(* POU Stations/ST_03_Ruestsaetze/ST_03_PRGs/ST03_Init_AbholPos, ST *)
PROGRAM ST03_Init_AbholPos
VAR
	RoboPos31		:BOOL;
	RoboPos35		:BOOL;
	RoboPosErr		:BOOL;
	CamDone			:BOOL;
	fb_Ton_PosErr	:TON;

	MsgOK			: BOOL;
END_VAR
(* Hier werden alle Abholpositionen am Rüstsatz bestimmt.
Ausnahmen:
	alte Rüstsätze:
		P360 74pol 
		P379 91pol 
		P489 168pol
		P4992 35pol
	Tampondrucker:
		P312 93pol
		P4991 102pol			*)

RoboPos31:=FALSE;
RoboPos35:=FALSE;
RoboPosErr:=FALSE;
CASE  gTypeCode OF

360,489:	(*74polig, 91polig, 168polig*)

	RoboPos31:=TRUE;

379: (*91 pol*)
RoboPos31:=
		ST08_412_B59_0.BitInToCheck;
	ST03_Main.Result:=RESULT_OK;		(* immer OK, wenn es keine Prüfung gibt*)

4992: (*35polig*)
	RoboPos31:=
		NOT ST08_412_B58_5_35pol.BitInToCheck AND	(*links*)
		ST08_412_B58_6_35pol.BitInToCheck;			(*rechts*)
	RoboPos35:=
		ST08_412_B58_5_35pol.BitInToCheck AND		(*links*)
		NOT ST08_412_B58_6_35pol.BitInToCheck;		(*rechts*)
	RoboPosErr:=
		ST08_412_B58_5_35pol.BitInToCheck AND		(*links*)
		ST08_412_B58_6_35pol.BitInToCheck;			(*rechts*)
	ST03_Main.Result:=RESULT_OK;		(* immer OK, wenn es keine Prüfung gibt*)

4871:(*154polig*)
	RoboPos31:=
		ST03_426_B68_4.BitInToCheck; 		(* Zuführung ISK auf Übergabeposition Robo Palettierer*)
	ST03_Main.Result:=RESULT_OK;		(* immer OK, wenn es keine Prüfung gibt*)

4872:(*154 Rasterplatte*)
	RoboPos31:=
			ST03_419_B61_2.BitInToCheck AND 	(*  Züführung links ISK auf Übergabeposition Roboter Palettierer*)
			ST03_419_B61_3.BitInToCheck;		(*  Züführung rechts ISK auf Übergabeposition Roboter Palettierer*)
	ST03_Main.Result:=RESULT_OK;			(* immer OK, wenn es keine Prüfung gibt*)

322: (*160polig*)
	RoboPos31:=
		ST03_422_B64_4.BitInToCheck; 			(* Zuführung ISK auf Übergabeposition Robo Palettierer*)

522:(*P522 206 polig*)
	RoboPos31:=
		ST03_437_B68_4.BitInToCheck AND
		NOT ST03_436_B68_1.BitInToCheck AND	(*links*)
		ST03_436_B68_2.BitInToCheck;			(*rechts*)
	RoboPos35:=
		ST03_437_B68_4.BitInToCheck AND
		ST03_436_B68_1.BitInToCheck AND		(*links*)
		NOT ST03_436_B68_2.BitInToCheck;		(*rechts*)
	RoboPosErr:=
(*		ST03_437_B68_4.BitInToCheck AND*)
		ST03_436_B68_1.BitInToCheck AND		(*links*)
		ST03_436_B68_2.BitInToCheck;		(*rechts*)
	ST03_Main.Result:=RESULT_OK;		(* immer OK, wenn es keine Prüfung gibt*)

550:(*P550 92 polig*)
	RoboPos31:=
		ST03_446_B70_4.BitInToCheck AND
		ST03_445_B70_1.BitInToCheck	AND		(*rechts*)
		NOT ST03_445_B70_2.BitInToCheck;			(*links*)
	RoboPos35:=
		ST03_446_B70_4.BitInToCheck AND
		NOT ST03_445_B70_1.BitInToCheck	AND	(*rechts*)
		ST03_445_B70_2.BitInToCheck;				(*links*)
	RoboPosErr:=
		ST03_446_B70_4.BitInToCheck AND
		ST03_445_B70_1.BitInToCheck AND	(*links*)
		ST03_445_B70_2.BitInToCheck;		(*rechts*)
	ST03_Main.Result:=RESULT_OK;		(* immer OK, wenn es keine Prüfung gibt*)

564:(*P564 124 polig*)
	RoboPos31:=
		ST03_453_B70_4.BitInToCheck AND
		ST03_452_B70_1.BitInToCheck	AND	(*rechts*)
		NOT	ST03_452_B70_2.BitInToCheck;	(*links*)
	RoboPos35:=
		ST03_453_B70_4.BitInToCheck AND
		NOT ST03_452_B70_1.BitInToCheck	AND	(*rechts*)
		ST03_452_B70_2.BitInToCheck;				(*links*)
	RoboPosErr:=
		ST03_446_B70_4.BitInToCheck AND
		ST03_445_B70_1.BitInToCheck AND	(*links*)
		ST03_445_B70_2.BitInToCheck;		(*rechts*)
	ST03_Main.Result:=RESULT_OK;		(* immer OK, wenn es keine Prüfung gibt*)

569:(*P569 46 polig*)
	RoboPos31:=
		ST03_463_B70_7.BitInToCheck AND
		ST03_462_B70_1.BitInToCheck	AND	(*rechts*)
		NOT	ST03_462_B70_2.BitInToCheck;	(*links*)
	RoboPos35:=
		ST03_463_B70_7.BitInToCheck AND
		NOT ST03_462_B70_1.BitInToCheck	AND(*rechts*)
		ST03_462_B70_2.BitInToCheck;
	RoboPosErr:=
		ST03_463_B70_7.BitInToCheck AND
		ST03_462_B70_1.BitInToCheck AND 	(*links*)
		ST03_462_B70_2.BitInToCheck;		(*rechts*)
	ST03_Main.Result:=RESULT_OK;		(* immer OK, wenn es keine Prüfung gibt*)

5731:(*P573 88polig*)
	RoboPos31:=
		ST03_501_B69_7. BitInToCheck AND	(*ISK auf Abholposition Robi*)
		NOT ST03_502_B70_0.BitInToCheck;	(*ISK Lageerkennung*)
	RoboPos35:=
		ST03_501_B69_7. BitInToCheck AND	(*ISK auf Abholposition Robi*)
		ST03_502_B70_0.BitInToCheck;		(*ISK Lageerkennung*)
	ST03_Main.Result:=RESULT_OK;		(* immer OK, wenn es keine Prüfung gibt*)

575,5753,5754,5755:(*P575 7polig*)
	RoboPos31:=
		ST03_513_B70_7.BitInToCheck AND		(*ISK auf Übergabeposition  1*)
		ST03_514_B71_2.BitInToCheck	AND	(*ISK auf Übergabeposition  2*)
		ST03_514_B71_5.BitInToCheck	AND	(*ISK auf Übergabeposition  3*)
		ST03_514_B71_6.BitInToCheck;			(*ISK auf Übergabeposition  4*)
	ST03_Main.Result:=RESULT_OK;			(* immer OK, wenn es keine Prüfung gibt*)

5732:(*P573 88polig AMG*)
	RoboPos31:=
		ST03_521_B69_7. BitInToCheck AND	(*ISK Lageerkennung links*)
		NOT ST03_522_B70_0.BitInToCheck;	(*ISK Lageerkennung rechts*)
	RoboPos35:=
		NOT ST03_521_B69_7. BitInToCheck AND(*ISK Lageerkennung links*)
		ST03_522_B70_0.BitInToCheck;			(*ISK Lageerkennung rechts*)
	RoboPosErr:=
		ST03_521_B69_7.BitInToCheck AND	(*links*)
		ST03_522_B70_0.BitInToCheck;		(*rechts*)
	ST03_Main.Result:=RESULT_OK;		(*immer OK, wenn es keine Prüfung gibt*)

5631:(*NOX 4pol*)
	RoboPos31:=
		ST03_491_B69_7.BitInToCheck;		(*Zuführung ISK auf Übergabeposition Robo Palettierer*)
	ST03_Main.Result:=RESULT_OK;		(*immer OK, wenn es keine Prüfung gibt*)

5632:(*NOX 5pol*)
	RoboPos31:=
		ST03_4x3_B70_0.BitInToCheck AND 	(*Pos 1*)		(* ISK anwesend Übergabeposition Stopper *)
		ST03_4x3_B70_1.BitInToCheck; (*AND	(*Pos 2*)		(* ISK anwesend Übergabeposition *)
		ST03_NOX_5pol_Zufuehrung.Result <> RESULT_NON; *)	(*warte bis Kamera fertig ist*)
	ST03_Main.Result:=ST03_NOX_5pol_Zufuehrung.Result;

5633:(*NOX 6pol*)
	RoboPos31:=
		ST03_4x3_B70_0.BitInToCheck AND 	(*Pos 1*)		(* ISK anwesend Übergabeposition Stopper *)
		ST03_4x3_B70_1.BitInToCheck AND	(*Pos 2*)		(* ISK anwesend Übergabeposition *)
		NOT ST03_NOX_6pol_Zufuehrung.LockForCam; 		(*warte bis Kamera fertig ist*)
	ST03_Main.Result:=ST03_NOX_6pol_Zufuehrung.Result;

5771:(*P5771 120polig*);
	RoboPos31:=
		ST03_531_B69_7. BitInToCheck AND	(*ISK rechts Lageerkennung*)
		NOT ST03_532_B70_0.BitInToCheck;	(*ISK links Lageerkennung*)
	RoboPos35:=
		NOT ST03_531_B69_7. BitInToCheck AND	(*ISK rechts Lageerkennung*)
		ST03_532_B70_0.BitInToCheck;		(*ISK links Lageerkennung*)
	RoboPosErr:=
		ST03_531_B69_7.BitInToCheck AND	(*links*)
		ST03_532_B70_0.BitInToCheck;		(*rechts*)

	ST03_Main.Result:=RESULT_OK;		(*immer OK, wenn es keine Prüfung gibt*)

5772:(*P5772 21polig*)
	RoboPos31:=
		NOT ST03_536_B69_7. BitInToCheck AND	(*ISK anwesend an Abholposition*)
		ST03_537_B70_0.BitInToCheck;	(*ISK Lageerkennung*)
	RoboPos35:=
		ST03_536_B69_7. BitInToCheck AND	(*ISK anwesend an Abholposition*)
		ST03_537_B70_0.BitInToCheck;		(*ISK Lageerkennung*)
	RoboPosErr:=
		ST03_536_B69_7.BitInToCheck AND			(*links*)
		NOT ST03_537_B70_0.BitInToCheck;		(*rechts*)
	ST03_Main.Result:=RESULT_OK;		(*immer OK, wenn es keine Prüfung gibt*)

580:(*P580 191polig*)
	RoboPos31:=
		ST03_541_B69_7. BitInToCheck AND		(*ISK links Lageerkennung*)
		NOT ST03_542_B70_0.BitInToCheck;		(*ISK rechts Lageerkennung*)
	RoboPos35:=
		NOT ST03_541_B69_7. BitInToCheck AND	(*ISK links Lageerkennung*)
		ST03_542_B70_0.BitInToCheck;				(*ISK rechts Lageerkennung*)
	RoboPosErr:=
		ST03_541_B69_7.BitInToCheck AND	(*links*)
		ST03_542_B70_0.BitInToCheck;		(*rechts*)
	ST03_Main.Result:=RESULT_OK;		(*immer OK, wenn es keine Prüfung gibt*)

5831:(*P5831 72polig*)
	RoboPos31:=
		ST03_546_B69_7. BitInToCheck AND		(*ISK rechts Lageerkennung*)
		NOT ST03_547_B70_0.BitInToCheck;		(*ISK links Lageerkennung*)
	RoboPos35:=
		NOT ST03_546_B69_7. BitInToCheck AND	(*ISK rechts Lageerkennung*)
		ST03_547_B70_0.BitInToCheck;				(*ISK links Lageerkennung*)
	RoboPosErr:=
		ST03_546_B69_7.BitInToCheck AND	(*links*)
		ST03_547_B70_0.BitInToCheck;		(*rechts*)
	ST03_Main.Result:=RESULT_OK;		(*immer OK, wenn es keine Prüfung gibt*)

5832:(*P5832 48polig*)
	RoboPos31:=
		ST03_551_B69_7. BitInToCheck AND		(*ISK rechts Lageerkennung*)
		NOT ST03_552_B70_0.BitInToCheck;		(*ISK links Lageerkennung*)
	RoboPos35:=
		NOT ST03_551_B69_7. BitInToCheck AND	(*ISK rechts Lageerkennung*)
		ST03_552_B70_0.BitInToCheck;				(*ISK links Lageerkennung*)
	RoboPosErr:=
		ST03_551_B69_7.BitInToCheck AND	(*links*)
		ST03_552_B70_0.BitInToCheck;		(*rechts*)
	ST03_Main.Result:=RESULT_OK;		(*immer OK, wenn es keine Prüfung gibt*)

5841, 4993:(*P5841 268pol, 102pol neu*)

	RoboPos31:=
		ST03_556_B69_7. BitInToCheck;		(*ISK anwesend an Abholposition*)

	ST03_Main.Result:=RESULT_OK;		(*immer OK, wenn es keine Prüfung gibt*)

5842:(*P584 268poligRP*)
	RoboPos31:=
	ST03_562_B67_7. BitInToCheck AND		(*Zuführung 1 ISK auf Übergabepos. Robi*)
	ST03_563_B70_7. BitInToCheck;			(*Zuführung 2 ISK auf Übergabepos. Robi*)
	ST03_Main.Result:=RESULT_OK;		(*immer OK, wenn es keine Prüfung gibt*)

598:(*P598 33polig*)

	RoboPos31:=
		ST03_571_B69_7. BitInToCheck;		(*ISK anwesend an Abholposition*)

	ST03_Main.Result:=RESULT_OK;		(*immer OK, wenn es keine Prüfung gibt*)

END_CASE

IF	RoboPos31 AND RoboPos35 THEN
	RoboPos31:=FALSE;
	RoboPos35:=FALSE;
END_IF


fb_Ton_PosErr(IN:=RoboPosErr,PT:=t#1s);
IF	ModeSelect.Mode>MODE_MANUAL AND fb_Ton_PosErr.Q THEN

	IF 	MessageHandler.Msg.ID <> 'PM122' THEN
		MessageHandler.ClearMessageLines(sVisu:=Visu.Message);
	END_IF
	MessageHandler.Msg.ID:='PM122';
	MessageHandler.Msg.Name:='Zuführung Lageerkennung';
	MessageHandler.Msg.Text:='Zuführung Lageerkennung prüfen';
	MessageHandler.Msg.Color:=Color.red;
	MessageHandler.Msg.Station:=0;

	MessageHandler(
		Prio:=2, 						(*1=highest, .. , 4=lowest*)
		Btn1Addr:=ADR(MsgOk),		(*Address of Button1 , if Zero then Button is unvisible*)
		Btn2Addr:=,					(*Address of Button2 , if Zero then Button is unvisible*)
		sVisu:=Visu.Message);

	IF 	MsgOK  OR NOT fb_Ton_PosErr.Q THEN
		MsgOk:=FALSE;
	END_IF

END_IF
END_PROGRAM

(* POU Stations/ST_03_Ruestsaetze/ST_03_SFCs/Zufuehrungen/ST03_NOX_5pol_Zufuehrung, SFC *)
 PROGRAM ST03_NOX_5pol_Zufuehrung
VAR_OUTPUT
	SFCCurrentPOU			: STRING:='ST03_NOX_5pol_Zufuehrung';
	SFCCurrentStep			: STRING:='';
	FB_CurrentStepHistorie	: FB_CurrentStepHistorie;
	SFCTime					: DINT;
	State   				: StateObject	:= STATE_WAIT;
	Result  				: StateResult;
END_VAR
VAR_INPUT
	Start				:BOOL;
END_VAR
VAR
	MsgOK				: BOOL;
	MsgCancel			: BOOL;
	SFCRun				: BOOL;
	SFCTimeStart		: TIME;
	Delay				: TON;
	(* Userdefinded area *)

	i					: INT;
	RepeatCounter		: INT;
	NokCounter			: INT;
	NokCounterPercent	: INT;
  	NokPercent   		: ARRAY[1..100] OF BOOL;
END_VAR
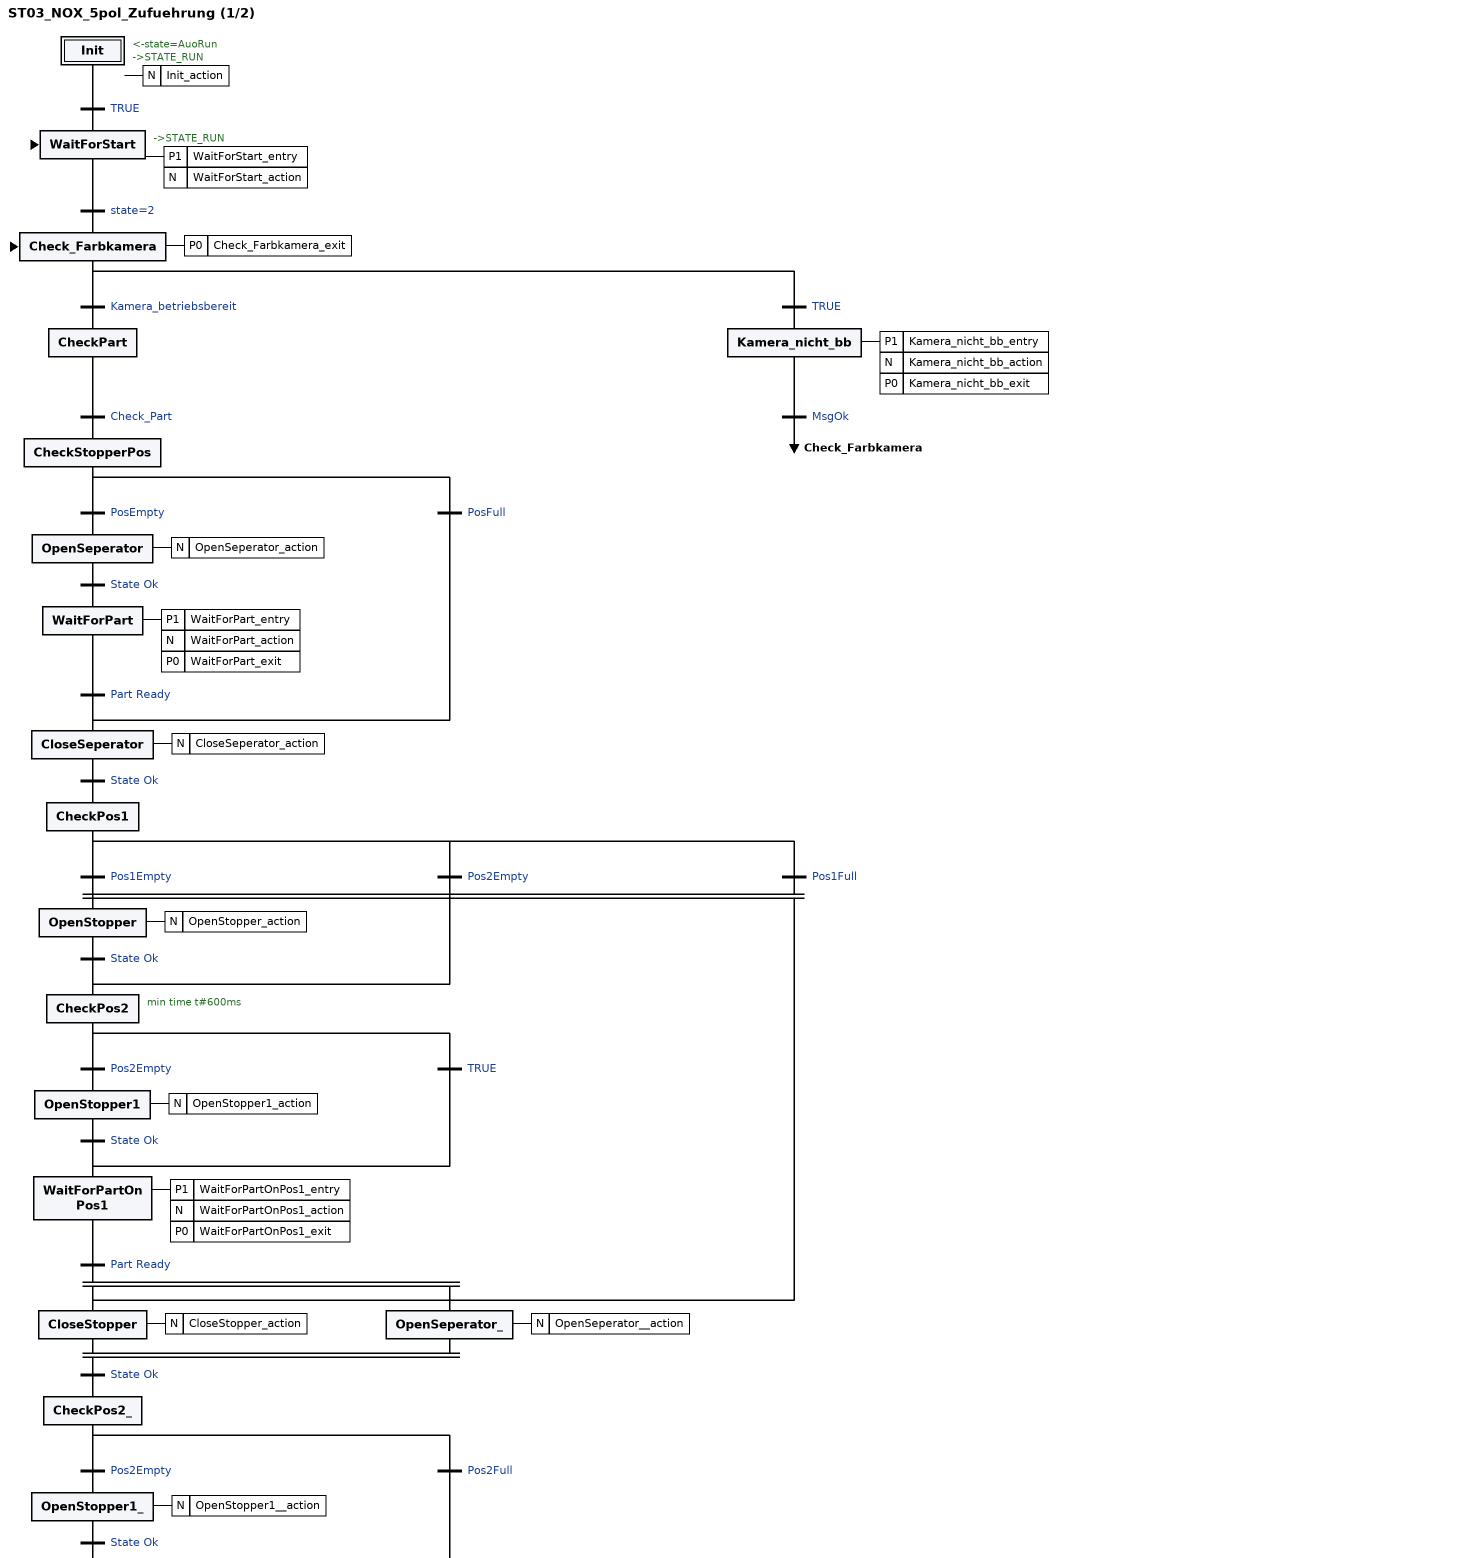
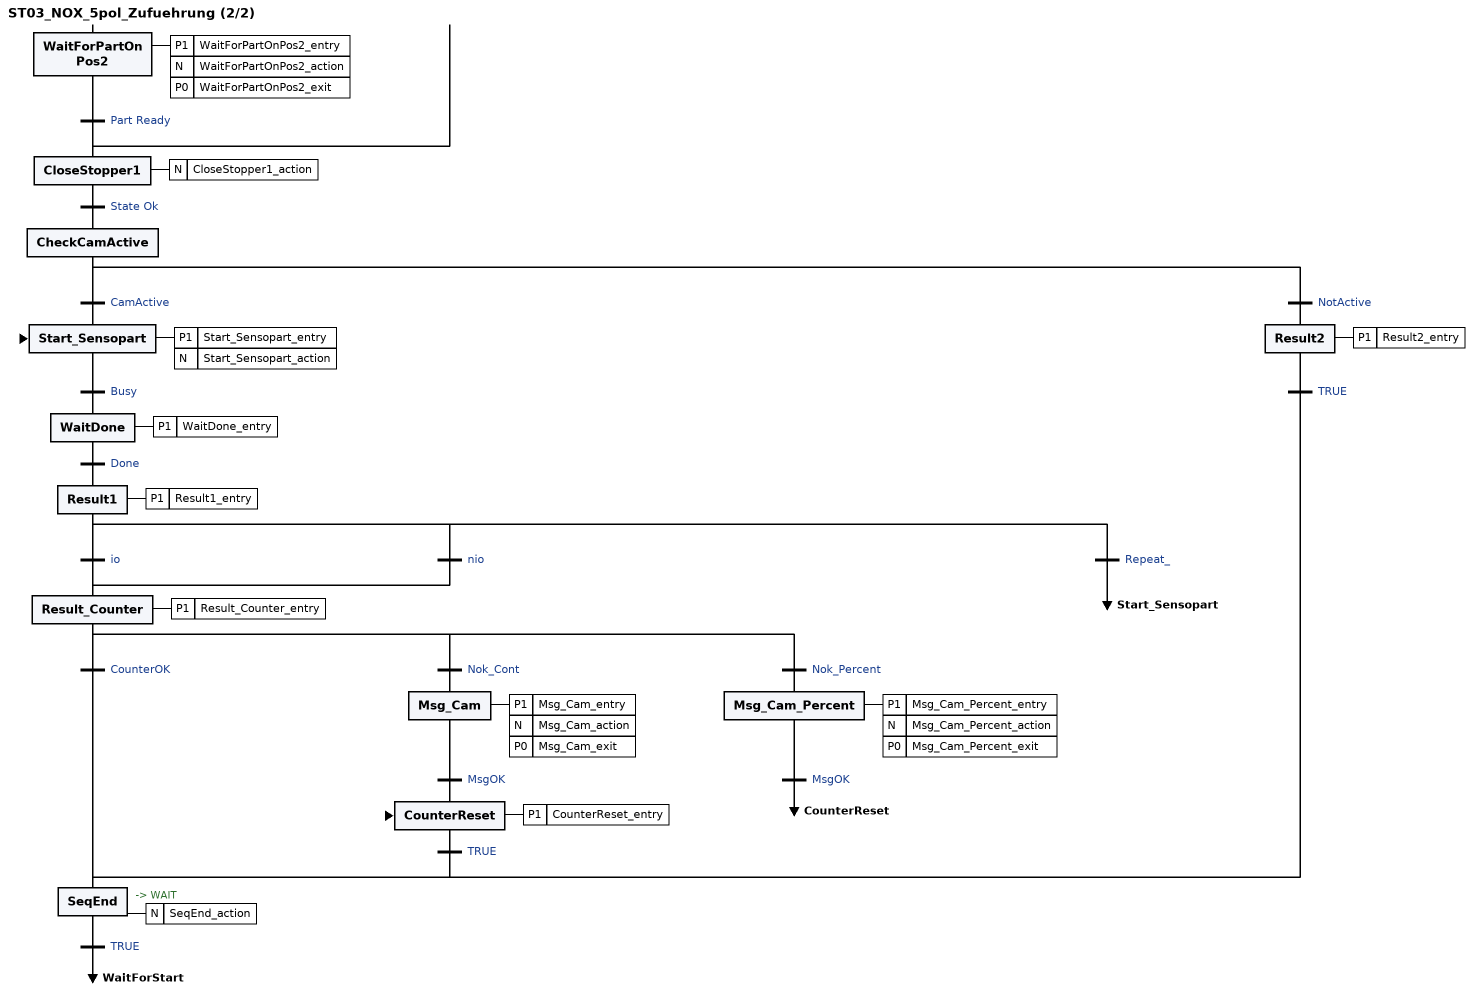
INITIAL_STEP Init: (* <-state=AuoRun / ->STATE_RUN *)
	Init_action(N);
END_STEP
TRANSITION FROM Init TO WaitForStart := TRUE;
END_TRANSITION
STEP WaitForStart: (* ->STATE_RUN *)
	WaitForStart_entry(P1);
	WaitForStart_action(N);
END_STEP
TRANSITION FROM WaitForStart TO Check_Farbkamera := state=2;
END_TRANSITION
STEP Check_Farbkamera:
	Check_Farbkamera_exit(P0);
END_STEP
TRANSITION FROM Check_Farbkamera TO CheckPart := Kamera_betriebsbereit;
END_TRANSITION
TRANSITION FROM Check_Farbkamera TO Kamera_nicht_bb := TRUE;
END_TRANSITION
STEP Kamera_nicht_bb:
	Kamera_nicht_bb_entry(P1);
	Kamera_nicht_bb_action(N);
	Kamera_nicht_bb_exit(P0);
END_STEP
TRANSITION FROM Kamera_nicht_bb TO Check_Farbkamera := MsgOk;
END_TRANSITION
STEP CheckPart:
END_STEP
TRANSITION FROM CheckPart TO CheckStopperPos := Check_Part;
END_TRANSITION
STEP CheckStopperPos:
END_STEP
TRANSITION FROM CheckStopperPos TO OpenSeperator := PosEmpty;
END_TRANSITION
TRANSITION FROM CheckStopperPos TO CloseSeperator := PosFull;
END_TRANSITION
STEP OpenSeperator:
	OpenSeperator_action(N);
END_STEP
TRANSITION FROM OpenSeperator TO WaitForPart := State Ok;
END_TRANSITION
STEP WaitForPart:
	WaitForPart_entry(P1);
	WaitForPart_action(N);
	WaitForPart_exit(P0);
END_STEP
TRANSITION FROM WaitForPart TO CloseSeperator := Part Ready;
END_TRANSITION
STEP CloseSeperator:
	CloseSeperator_action(N);
END_STEP
TRANSITION FROM CloseSeperator TO CheckPos1 := State Ok;
END_TRANSITION
STEP CheckPos1:
END_STEP
TRANSITION FROM CheckPos1 TO OpenStopper := Pos1Empty;
END_TRANSITION
TRANSITION FROM CheckPos1 TO CheckPos2 := Pos2Empty;
END_TRANSITION
TRANSITION FROM CheckPos1 TO (CloseStopper, OpenSeperator_) := Pos1Full;
END_TRANSITION
STEP OpenStopper:
	OpenStopper_action(N);
END_STEP
TRANSITION FROM OpenStopper TO CheckPos2 := State Ok;
END_TRANSITION
STEP CheckPos2: (* min time t#600ms *)
END_STEP
TRANSITION FROM CheckPos2 TO OpenStopper1 := Pos2Empty;
END_TRANSITION
TRANSITION FROM CheckPos2 TO WaitForPartOnPos1 := TRUE;
END_TRANSITION
STEP OpenStopper1:
	OpenStopper1_action(N);
END_STEP
TRANSITION FROM OpenStopper1 TO WaitForPartOnPos1 := State Ok;
END_TRANSITION
STEP WaitForPartOnPos1:
	WaitForPartOnPos1_entry(P1);
	WaitForPartOnPos1_action(N);
	WaitForPartOnPos1_exit(P0);
END_STEP
TRANSITION FROM WaitForPartOnPos1 TO (CloseStopper, OpenSeperator_) := Part Ready;
END_TRANSITION
STEP CloseStopper:
	CloseStopper_action(N);
END_STEP
STEP OpenSeperator_:
	OpenSeperator__action(N);
END_STEP
TRANSITION FROM (CloseStopper, OpenSeperator_) TO CheckPos2_ := State Ok;
END_TRANSITION
STEP CheckPos2_:
END_STEP
TRANSITION FROM CheckPos2_ TO OpenStopper1_ := Pos2Empty;
END_TRANSITION
TRANSITION FROM CheckPos2_ TO CloseStopper1 := Pos2Full;
END_TRANSITION
STEP OpenStopper1_:
	OpenStopper1__action(N);
END_STEP
TRANSITION FROM OpenStopper1_ TO WaitForPartOnPos2 := State Ok;
END_TRANSITION
STEP WaitForPartOnPos2:
	WaitForPartOnPos2_entry(P1);
	WaitForPartOnPos2_action(N);
	WaitForPartOnPos2_exit(P0);
END_STEP
TRANSITION FROM WaitForPartOnPos2 TO CloseStopper1 := Part Ready;
END_TRANSITION
STEP CloseStopper1:
	CloseStopper1_action(N);
END_STEP
TRANSITION FROM CloseStopper1 TO CheckCamActive := State Ok;
END_TRANSITION
STEP CheckCamActive:
END_STEP
TRANSITION FROM CheckCamActive TO Start_Sensopart := CamActive;
END_TRANSITION
TRANSITION FROM CheckCamActive TO Result2 := NotActive;
END_TRANSITION
STEP Start_Sensopart:
	Start_Sensopart_entry(P1);
	Start_Sensopart_action(N);
END_STEP
TRANSITION FROM Start_Sensopart TO WaitDone := Busy;
END_TRANSITION
STEP WaitDone:
	WaitDone_entry(P1);
END_STEP
TRANSITION FROM WaitDone TO Result1 := Done;
END_TRANSITION
STEP Result1:
	Result1_entry(P1);
END_STEP
TRANSITION FROM Result1 TO Result_Counter := io;
END_TRANSITION
TRANSITION FROM Result1 TO Result_Counter := nio;
END_TRANSITION
TRANSITION FROM Result1 TO Start_Sensopart := Repeat_;
END_TRANSITION
STEP Result_Counter:
	Result_Counter_entry(P1);
END_STEP
TRANSITION FROM Result_Counter TO SeqEnd := CounterOK;
END_TRANSITION
TRANSITION FROM Result_Counter TO Msg_Cam := Nok_Cont;
END_TRANSITION
TRANSITION FROM Result_Counter TO Msg_Cam_Percent := Nok_Percent;
END_TRANSITION
STEP Msg_Cam:
	Msg_Cam_entry(P1);
	Msg_Cam_action(N);
	Msg_Cam_exit(P0);
END_STEP
TRANSITION FROM Msg_Cam TO CounterReset := MsgOK;
END_TRANSITION
STEP CounterReset:
	CounterReset_entry(P1);
END_STEP
TRANSITION FROM CounterReset TO SeqEnd := TRUE;
END_TRANSITION
STEP Msg_Cam_Percent:
	Msg_Cam_Percent_entry(P1);
	Msg_Cam_Percent_action(N);
	Msg_Cam_Percent_exit(P0);
END_STEP
TRANSITION FROM Msg_Cam_Percent TO CounterReset := MsgOK;
END_TRANSITION
STEP Result2:
	Result2_entry(P1);
END_STEP
TRANSITION FROM Result2 TO SeqEnd := TRUE;
END_TRANSITION
STEP SeqEnd: (* -> WAIT *)
	SeqEnd_action(N);
END_STEP
TRANSITION FROM SeqEnd TO WaitForStart := TRUE;
END_TRANSITION

ACTION Init_action:
Start:=FALSE;
State:=STATE_WAIT;
MsgOK:=FALSE;
MsgCancel:=FALSE;
SFCRun:=FALSE;
Result:=RESULT_NON;
END_ACTION

ACTION WaitForStart_entry:
;
END_ACTION

ACTION WaitForStart_action:
IF 	Start   THEN
	State:=STATE_RUN;
	SFCTimeStart:=TIME();
	Start:=FALSE;
ELSE
	State:=STATE_WAIT;
	MsgOK:=FALSE;
	MsgCancel:=FALSE;
	SFCRun:=FALSE;
END_IF
END_ACTION

ACTION Check_Farbkamera_exit:
Result:=RESULT_NON;

IF NOT ST03_8_100_A1.Activated THEN
	Result:= RESULT_OK;
END_IF
END_ACTION

ACTION Kamera_nicht_bb_entry:
MessageHandler.ClearMessageLines(sVisu:=Visu.Message);
END_ACTION

ACTION Kamera_nicht_bb_action:
MessageHandler.Msg.ID:='PM152';
MessageHandler.Msg.Name:='Check Camera';
MessageHandler.Msg.Text:='Sesopart Kamera ist nicht betriebsbereit';
MessageHandler.Msg.Color:=Color.red;
MessageHandler.Msg.Station:=1;


MessageHandler(
	Prio:=2, 							(*1=highest, .. , 4=lowest*)
	Btn1Addr:=ADR(MsgOk),			(*Address of Button1 , if Zero then Button is unvisible*)
	Btn2Addr:=,						(*Address of Button2 , if Zero then Button is unvisible*)
	sVisu:=Visu.Message);
END_ACTION

ACTION Kamera_nicht_bb_exit:
MsgOk:=FALSE;
MsgCancel:=FALSE;
ST02_DT_95_A1.b_quitt:=TRUE;
END_ACTION

ACTION OpenSeperator_action:
ST03_4x3_Y70_5.MoveInit:=TRUE;		(*Zuführung Vereinzler AST/GST *)
END_ACTION

ACTION WaitForPart_entry:
ProcessMessage02:='';
Delay(IN:=FALSE);
END_ACTION

ACTION WaitForPart_action:
ProcessMessage02:='2IM6';				(*warte auf Teil Übergabeposition 1*)
Delay(	IN:=ST03_4x2_B69_5.BitInToCheck, (*ISK anwesend am Stopper*)
		PT:=T#50ms);
END_ACTION

ACTION WaitForPart_exit:
ProcessMessage02:='';
END_ACTION

ACTION CloseSeperator_action:
ST03_4x3_Y70_5.MoveWork:=TRUE;		(*Zuführung Vereinzler AST/GST *)
END_ACTION

ACTION OpenStopper_action:
ST03_4x3_Y70_6.MoveWork:=TRUE;		(*Zuführung Stopper AST/GST *)
END_ACTION

ACTION OpenStopper1_action:
ST03_4x3_Y70_7.MoveWork:=TRUE;		(* Zuführung Stopper Übergabeposition AST/GST*)
END_ACTION

ACTION WaitForPartOnPos1_entry:
ProcessMessage02:='';
Delay(IN:=FALSE);
END_ACTION

ACTION WaitForPartOnPos1_action:
ProcessMessage02:='2IM6';					(*warte auf Teil Übergabeposition 1*)
Delay.IN:=ST03_4x3_B70_0.BitInToCheck;  	(*ISK anwesend Übergabeposition Stopper *)

Delay.PT:=T#50ms;
Delay();
END_ACTION

ACTION WaitForPartOnPos1_exit:
ProcessMessage02:='';
END_ACTION

ACTION CloseStopper_action:
ST03_4x3_Y70_6.MoveInit:=TRUE;		(*Zuführung Stopper AST/GST *)
END_ACTION

ACTION OpenSeperator__action:
ST03_4x3_Y70_5.MoveInit:=TRUE;		(*Zuführung Vereinzler AST/GST *)
END_ACTION

ACTION OpenStopper1__action:
ST03_4x3_Y70_7.MoveWork:=TRUE;		(* Zuführung Stopper Übergabeposition AST/GST*)
END_ACTION

ACTION WaitForPartOnPos2_entry:
ProcessMessage02:='';
Delay(IN:=FALSE);
END_ACTION

ACTION WaitForPartOnPos2_action:
ProcessMessage02:='2IM5';						(*warte auf Teil Übergabeposition 2*)
Delay(	IN:=ST03_4x3_B70_1.BitInToCheck, 		(*ISK anwesend Übergabeposition *)
		PT:=T#50ms);
END_ACTION

ACTION WaitForPartOnPos2_exit:
ProcessMessage02:='';
END_ACTION

ACTION CloseStopper1_action:
ST03_4x3_Y70_7.MoveInit:=TRUE;		(* Zuführung Stopper Übergabeposition AST/GST *)
END_ACTION

ACTION Start_Sensopart_entry:
Result:=RESULT_NON;
END_ACTION

ACTION Start_Sensopart_action:
ST03_8_100_A1.JobNo := TD.Sensopart_CamProgNo ;
ST03_8_100_A1.st_ctrl_in.b_start := TRUE;
END_ACTION

ACTION WaitDone_entry:
ST03_8_100_A1.st_ctrl_in.b_start := FALSE;
RepeatCounter:=RepeatCounter+1;
END_ACTION

ACTION Result1_entry:
IF 	(ST03_8_100_A1.b_Kam_Pruef_IO AND	 (*Kamera Farberkennung*)
	NOT ST03_8_100_A1.b_Kam_Pruef_NIO)THEN
	Result:=RESULT_OK;
ELSE
	Result:=RESULT_NOK;
END_IF
END_ACTION

ACTION Result_Counter_entry:
IF 	(ST02_DT_95_A2.b_Kam_Pruef_IO AND	 (*Kamera Farberkennung*)
	NOT ST02_DT_95_A2.b_Kam_Pruef_NIO)THEN
	Result:=Result+10;
ELSE
	Result:=Result+90;
END_IF

FOR i:=100 TO 2 BY-1 DO
   NokPercent[i] := NokPercent[i-1];
END_FOR

IF	Result = 11 THEN
	NokCounter:=0;
	NokPercent[1] := FALSE;
	gRob01GripState:=PART_OK;
ELSE
	NokCounter:=NokCounter+1;
	NokPercent[1] := TRUE;
	gRob01GripState:=PART_NOK;
END_IF
END_ACTION

ACTION Msg_Cam_entry:
MessageHandler.ClearMessageLines(sVisu:=Visu.Message);
END_ACTION

ACTION Msg_Cam_action:
MessageHandler.Msg.ID:='PM112';
MessageHandler.Msg.Name:='Sensopart Kam.-Erg. Prüfung  n.i.o:';
MessageHandler.Msg.Text:='Sensopart Kam.-Erg. Prüfung  n.i.o: Fehler in Folge';
MessageHandler.Msg.Color:=Color.red;
MessageHandler.Msg.Station:=3;
MessageHandler.MsgButton1Text:='continue';

MessageHandler(
	Prio:=2, 								(*1=highest, .. , 4=lowest*)
	Btn1Addr:=ADR(MsgOk),				(*Address of Button1 , if Zero then Button is unvisible*)
	Btn2Addr:=0(*ADR(MsgCancel)*),			(*Address of Button2 , if Zero then Button is unvisible*)
	sVisu:=Visu.Message);
END_ACTION

ACTION Msg_Cam_exit:
MsgOk:=FALSE;
MsgCancel:=FALSE;
END_ACTION

ACTION CounterReset_entry:
NokCounter:=0;
(*Percent Register löschen*)
FOR i:=1 TO 100 BY 1 DO
  NokPercent[i]:= FALSE;
END_FOR
END_ACTION

ACTION Msg_Cam_Percent_entry:
MessageHandler.ClearMessageLines(sVisu:=Visu.Message);
END_ACTION

ACTION Msg_Cam_Percent_action:
MessageHandler.Msg.ID:='PM113';
MessageHandler.Msg.Name:='Sensopart Kam.-Erg. Prüfung  n.i.o:';
MessageHandler.Msg.Text:='Sensopart Kam.-Erg. Prüfung  n.i.o:% Fehler';
MessageHandler.Msg.Color:=Color.red;
MessageHandler.Msg.Station:=3;
MessageHandler.MsgButton1Text:='continue';

MessageHandler(
	Prio:=2, 								(*1=highest, .. , 4=lowest*)
	Btn1Addr:=ADR(MsgOk),				(*Address of Button1 , if Zero then Button is unvisible*)
	Btn2Addr:=0(*ADR(MsgCancel)*),			(*Address of Button2 , if Zero then Button is unvisible*)
	sVisu:=Visu.Message);
END_ACTION

ACTION Msg_Cam_Percent_exit:
MsgOk:=FALSE;
MsgCancel:=FALSE;
END_ACTION

ACTION Result2_entry:
Result:= RESULT_OK;
END_ACTION

ACTION SeqEnd_action:
SFCTime:=TIME_TO_DINT(TIME()-SFCTimeStart);
State:=STATE_WAIT;
END_ACTION

TRANSITION Kamera_betriebsbereit:
(*Kamera Farberkennung*)
(
NOT ST03_8_100_A1.sm_kamera_nicht_bb OR
NOT ST03_8_100_A1.Activated	)
END_TRANSITION

TRANSITION Check_Part:
Robot01.ActualArea <> 4 AND
(
NOT ST03_4x3_B70_0.BitInToCheck OR	(* ISK anwesend Übergabeposition Stopper*)
NOT ST03_4x3_B70_1.BitInToCheck )	(* ISK anwesend Übergabeposition*)
END_TRANSITION

TRANSITION PosEmpty:
NOT ST03_4x2_B69_5.BitInToCheck			 	(*  ISK anwesend am Stopper*)
END_TRANSITION

TRANSITION State Ok:
ST03_4x3_Y70_5.State=STATE_OK (*Zuführung Vereinzler AST/GST *)
END_TRANSITION

TRANSITION Part Ready:
Delay.Q
END_TRANSITION

TRANSITION PosFull:
ST03_4x2_B69_5.BitInToCheck			 	(*  ISK anwesend am Stopper*)
END_TRANSITION

TRANSITION State Ok:
ST03_4x3_Y70_5.State=STATE_OK (*Zuführung Vereinzler AST/GST *)
END_TRANSITION

TRANSITION Pos1Empty:
NOT ST03_4x3_B70_0.BitInToCheck AND 	(*  ISK anwesend Übergabeposition Stopper*)
ST03_4x2_B69_5.BitInToCheck			 	(*  ISK anwesend am Stopper*)
END_TRANSITION

TRANSITION Pos2Empty:
ST03_4x3_B70_0.BitInToCheck AND 	(*  ISK anwesend Übergabeposition Stopper*)
NOT ST03_4x3_B70_1.BitInToCheck AND 	(*  ISK anwesend Übergabeposition*)
ST03_4x2_B69_5.BitInToCheck			 	(*  ISK anwesend am Stopper*)
END_TRANSITION

TRANSITION State Ok:
ST03_4x3_Y70_6.State=STATE_OK 	(*Zuführung Stopper AST/GST *)
END_TRANSITION

TRANSITION Pos2Empty:
NOT ST03_4x3_B70_1.BitInToCheck AND 	(*  ISK anwesend Übergabeposition*)
NOT ST03_4x2_B69_5.BitInToCheck			 (*ISK anwesend am Stopper*)
END_TRANSITION

TRANSITION State Ok:
ST03_4x3_Y70_7.State=STATE_OK 	(* Zuführung Stopper Übergabeposition AST/GST *)
END_TRANSITION

TRANSITION Part Ready:
Delay.Q
END_TRANSITION

TRANSITION Pos1Full:
ST03_4x3_B70_0.BitInToCheck 	(*ISK anwesend Übergabeposition Stopper*)
END_TRANSITION

TRANSITION State Ok:
ST03_4x3_Y70_6.State=STATE_OK AND	(*Zuführung Stopper AST/GST *)
ST03_4x3_Y70_5.State=STATE_OK (*Zuführung Vereinzler AST/GST *)
END_TRANSITION

TRANSITION Pos2Empty:
NOT ST03_4x3_B70_1.BitInToCheck AND 	(*  ISK anwesend Übergabeposition*)
ST03_4x3_B70_0.BitInToCheck			 	(*  ISK anwesend Übergabeposition Stopper*)
END_TRANSITION

TRANSITION State Ok:
ST03_4x3_Y70_7.State=STATE_OK 	(* Zuführung Stopper Übergabeposition AST/GST *)
END_TRANSITION

TRANSITION Part Ready:
Delay.Q
END_TRANSITION

TRANSITION Pos2Full:
ST03_4x3_B70_1.BitInToCheck	 	(*ISK anwesend Übergabeposition*)
END_TRANSITION

TRANSITION State Ok:
ST03_4x3_Y70_7.State=STATE_OK 	(* Zuführung Stopper Übergabeposition AST/GST *)
END_TRANSITION

TRANSITION CamActive:
ST03_8_100_A1.Activated
END_TRANSITION

TRANSITION Busy:
ST03_8_100_A1.st_ctrl_out.b_busy (*Kamera Farberkennung Ehternet*)
END_TRANSITION

TRANSITION Done:
ST03_8_100_A1.st_ctrl_out.b_fertig
END_TRANSITION

TRANSITION io:
Result = RESULT_OK
END_TRANSITION

TRANSITION nio:
RepeatCounter>=2
END_TRANSITION

TRANSITION Repeat_:
TRUE
END_TRANSITION

TRANSITION CounterOK:
NokCounter<MP.ST03.CamNoOfErrors AND
NokCounterPercent < MP.ST02.CamNoOfErrorsPercent
END_TRANSITION

TRANSITION Nok_Cont:
NokCounter >= MP.ST03.CamNoOfErrors
END_TRANSITION

TRANSITION Nok_Percent:
NokCounterPercent >= MP.ST03.CamNoOfErrorsPercent
END_TRANSITION

TRANSITION NotActive:
TRUE
END_TRANSITION
END_PROGRAM

(* POU Stations/ST_03_Ruestsaetze/ST_03_SFCs/Zufuehrungen/ST03_NOX_6pol_Zufuehrung, SFC *)
 PROGRAM ST03_NOX_6pol_Zufuehrung

VAR_OUTPUT
	SFCCurrentPOU			: STRING:='ST03_NOX_6pol_Zufuehrung';
	SFCCurrentStep			: STRING:='';
	FB_CurrentStepHistorie	: FB_CurrentStepHistorie;
	SFCTime					: DINT;
	State   				: StateObject	:= STATE_WAIT;
	Result  				: StateResult;
	LockForCam				: BOOL;

END_VAR
VAR_INPUT
	Start					: BOOL;
END_VAR
VAR
	MsgOK					: BOOL;
	MsgCancel				: BOOL;
	SFCRun					: BOOL;
	SFCTimeStart			: TIME;
	Delay					: TON;
	(* Userdefinded area *)

	i						: INT;
	RepeatCounter			: INT;
	NokCounter_Cam			: ARRAY[1..2] OF INT;
	NokCounterPercent_Cam	: ARRAY[1..2] OF INT;
  	NokPercent_Cam  		: ARRAY[1..2, 1..100] OF BOOL;

	Result_Cam1				: ARRAY[1..2] OF StateResult;
	Result_Cam2				: StateResult;
	Part					: INT := 0;	(*Teil 1 oder Teil 2*)

	KeyenceCam_AlwaysOK		: BOOL:=FALSE; (*Keyence RESULT_OK - nur für IBN*)
	SensopartCam_AlwaysOK	: BOOL:=FALSE; (*Sensopart RESULT_OK - nur für IBN*)
END_VAR
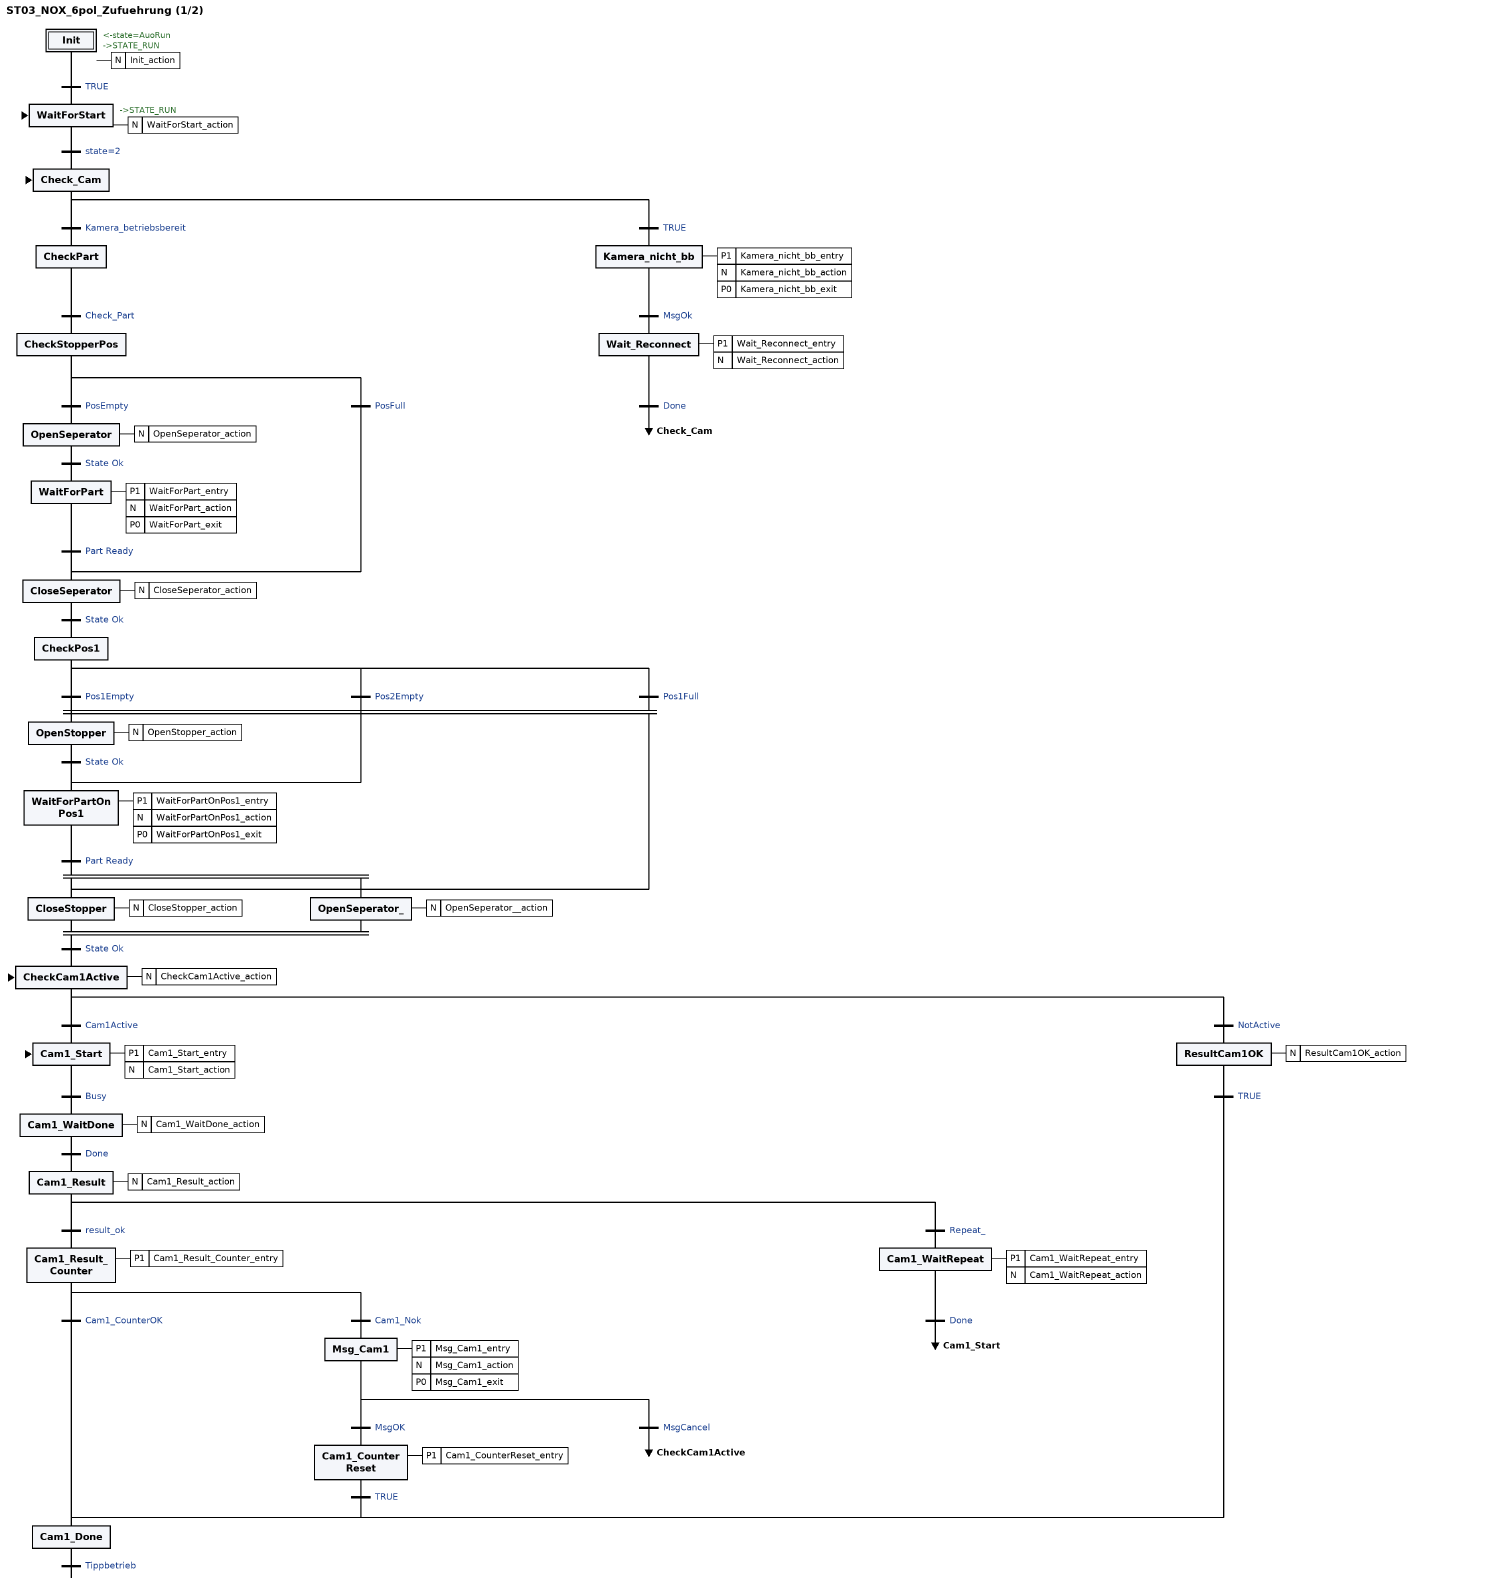
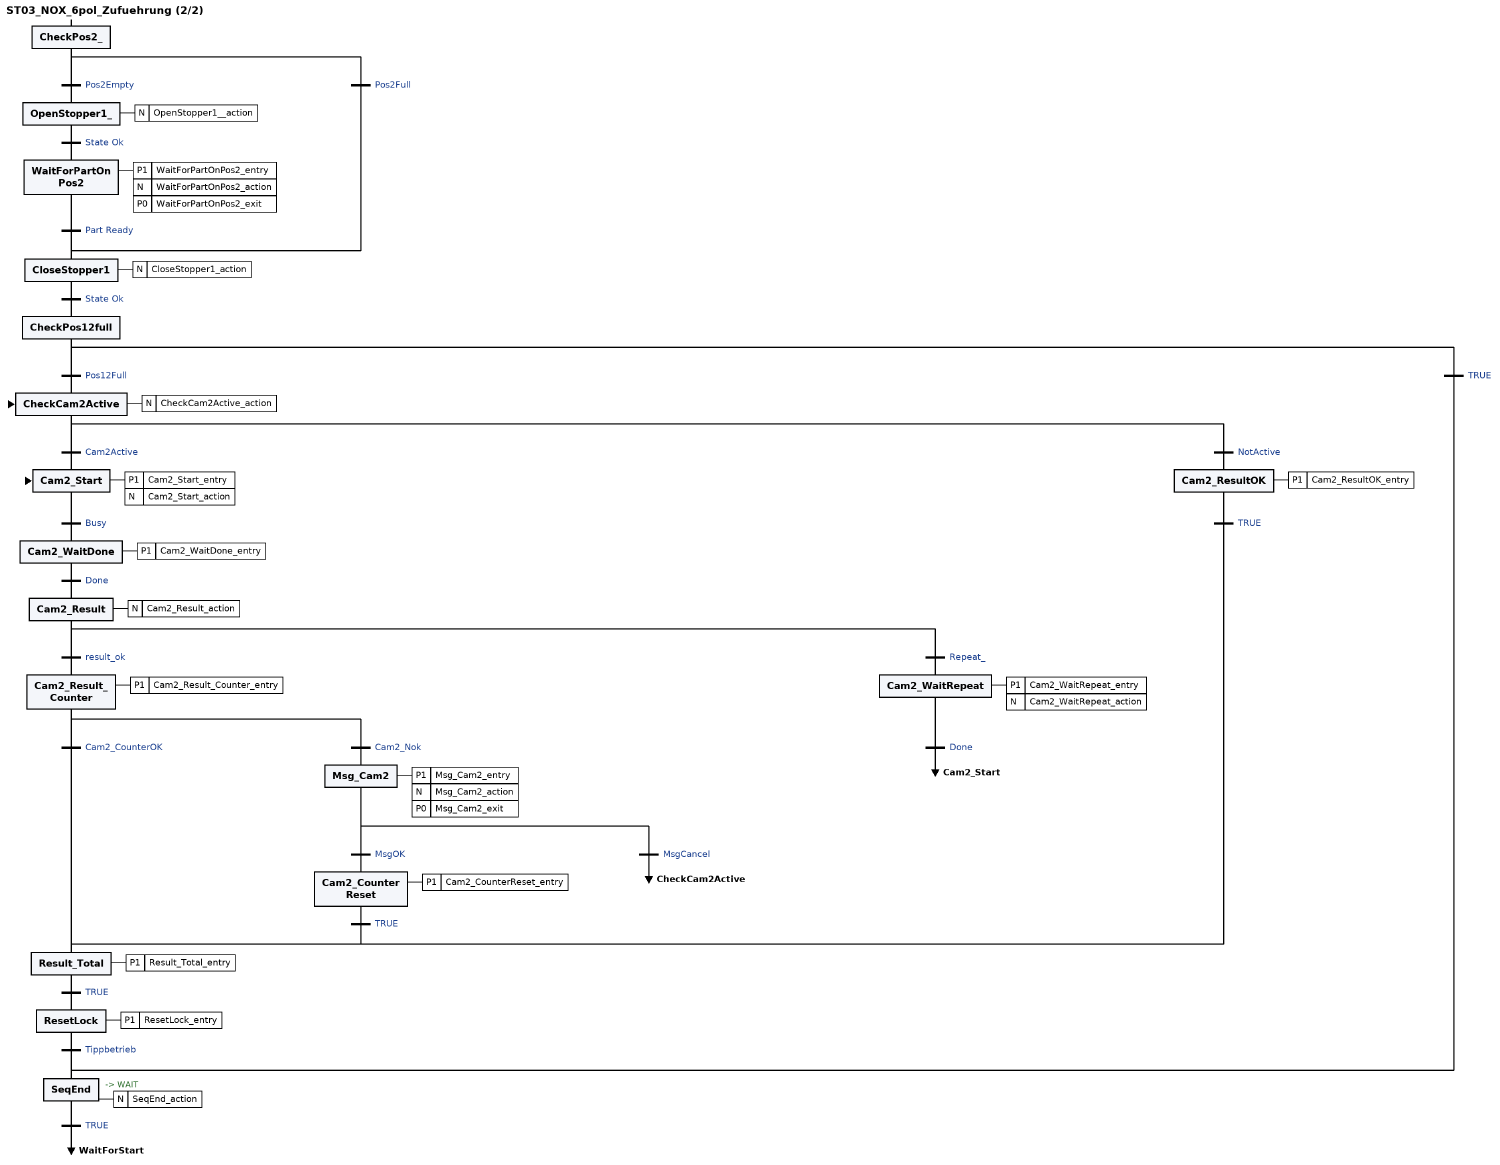
INITIAL_STEP Init: (* <-state=AuoRun / ->STATE_RUN *)
	Init_action(N);
END_STEP
TRANSITION FROM Init TO WaitForStart := TRUE;
END_TRANSITION
STEP WaitForStart: (* ->STATE_RUN *)
	WaitForStart_action(N);
END_STEP
TRANSITION FROM WaitForStart TO Check_Cam := state=2;
END_TRANSITION
STEP Check_Cam:
END_STEP
TRANSITION FROM Check_Cam TO CheckPart := Kamera_betriebsbereit;
END_TRANSITION
TRANSITION FROM Check_Cam TO Kamera_nicht_bb := TRUE;
END_TRANSITION
STEP Kamera_nicht_bb:
	Kamera_nicht_bb_entry(P1);
	Kamera_nicht_bb_action(N);
	Kamera_nicht_bb_exit(P0);
END_STEP
TRANSITION FROM Kamera_nicht_bb TO Wait_Reconnect := MsgOk;
END_TRANSITION
STEP Wait_Reconnect:
	Wait_Reconnect_entry(P1);
	Wait_Reconnect_action(N);
END_STEP
TRANSITION FROM Wait_Reconnect TO Check_Cam := Done;
END_TRANSITION
STEP CheckPart:
END_STEP
TRANSITION FROM CheckPart TO CheckStopperPos := Check_Part;
END_TRANSITION
STEP CheckStopperPos:
END_STEP
TRANSITION FROM CheckStopperPos TO OpenSeperator := PosEmpty;
END_TRANSITION
TRANSITION FROM CheckStopperPos TO CloseSeperator := PosFull;
END_TRANSITION
STEP OpenSeperator:
	OpenSeperator_action(N);
END_STEP
TRANSITION FROM OpenSeperator TO WaitForPart := State Ok;
END_TRANSITION
STEP WaitForPart:
	WaitForPart_entry(P1);
	WaitForPart_action(N);
	WaitForPart_exit(P0);
END_STEP
TRANSITION FROM WaitForPart TO CloseSeperator := Part Ready;
END_TRANSITION
STEP CloseSeperator:
	CloseSeperator_action(N);
END_STEP
TRANSITION FROM CloseSeperator TO CheckPos1 := State Ok;
END_TRANSITION
STEP CheckPos1:
END_STEP
TRANSITION FROM CheckPos1 TO OpenStopper := Pos1Empty;
END_TRANSITION
TRANSITION FROM CheckPos1 TO WaitForPartOnPos1 := Pos2Empty;
END_TRANSITION
TRANSITION FROM CheckPos1 TO (CloseStopper, OpenSeperator_) := Pos1Full;
END_TRANSITION
STEP OpenStopper:
	OpenStopper_action(N);
END_STEP
TRANSITION FROM OpenStopper TO WaitForPartOnPos1 := State Ok;
END_TRANSITION
STEP WaitForPartOnPos1:
	WaitForPartOnPos1_entry(P1);
	WaitForPartOnPos1_action(N);
	WaitForPartOnPos1_exit(P0);
END_STEP
TRANSITION FROM WaitForPartOnPos1 TO (CloseStopper, OpenSeperator_) := Part Ready;
END_TRANSITION
STEP CloseStopper:
	CloseStopper_action(N);
END_STEP
STEP OpenSeperator_:
	OpenSeperator__action(N);
END_STEP
TRANSITION FROM (CloseStopper, OpenSeperator_) TO CheckCam1Active := State Ok;
END_TRANSITION
STEP CheckCam1Active:
	CheckCam1Active_action(N);
END_STEP
TRANSITION FROM CheckCam1Active TO Cam1_Start := Cam1Active;
END_TRANSITION
TRANSITION FROM CheckCam1Active TO ResultCam1OK := NotActive;
END_TRANSITION
STEP Cam1_Start:
	Cam1_Start_entry(P1);
	Cam1_Start_action(N);
END_STEP
TRANSITION FROM Cam1_Start TO Cam1_WaitDone := Busy;
END_TRANSITION
STEP Cam1_WaitDone:
	Cam1_WaitDone_action(N);
END_STEP
TRANSITION FROM Cam1_WaitDone TO Cam1_Result := Done;
END_TRANSITION
STEP Cam1_Result:
	Cam1_Result_action(N);
END_STEP
TRANSITION FROM Cam1_Result TO Cam1_Result_Counter := result_ok;
END_TRANSITION
TRANSITION FROM Cam1_Result TO Cam1_WaitRepeat := Repeat_;
END_TRANSITION
STEP Cam1_WaitRepeat:
	Cam1_WaitRepeat_entry(P1);
	Cam1_WaitRepeat_action(N);
END_STEP
TRANSITION FROM Cam1_WaitRepeat TO Cam1_Start := Done;
END_TRANSITION
STEP Cam1_Result_Counter:
	Cam1_Result_Counter_entry(P1);
END_STEP
TRANSITION FROM Cam1_Result_Counter TO Cam1_Done := Cam1_CounterOK;
END_TRANSITION
TRANSITION FROM Cam1_Result_Counter TO Msg_Cam1 := Cam1_Nok;
END_TRANSITION
STEP Msg_Cam1:
	Msg_Cam1_entry(P1);
	Msg_Cam1_action(N);
	Msg_Cam1_exit(P0);
END_STEP
TRANSITION FROM Msg_Cam1 TO Cam1_CounterReset := MsgOK;
END_TRANSITION
TRANSITION FROM Msg_Cam1 TO CheckCam1Active := MsgCancel;
END_TRANSITION
STEP Cam1_CounterReset:
	Cam1_CounterReset_entry(P1);
END_STEP
TRANSITION FROM Cam1_CounterReset TO Cam1_Done := TRUE;
END_TRANSITION
STEP ResultCam1OK:
	ResultCam1OK_action(N);
END_STEP
TRANSITION FROM ResultCam1OK TO Cam1_Done := TRUE;
END_TRANSITION
STEP Cam1_Done:
END_STEP
TRANSITION FROM Cam1_Done TO CheckPos2_ := Tippbetrieb;
END_TRANSITION
STEP CheckPos2_:
END_STEP
TRANSITION FROM CheckPos2_ TO OpenStopper1_ := Pos2Empty;
END_TRANSITION
TRANSITION FROM CheckPos2_ TO CloseStopper1 := Pos2Full;
END_TRANSITION
STEP OpenStopper1_:
	OpenStopper1__action(N);
END_STEP
TRANSITION FROM OpenStopper1_ TO WaitForPartOnPos2 := State Ok;
END_TRANSITION
STEP WaitForPartOnPos2:
	WaitForPartOnPos2_entry(P1);
	WaitForPartOnPos2_action(N);
	WaitForPartOnPos2_exit(P0);
END_STEP
TRANSITION FROM WaitForPartOnPos2 TO CloseStopper1 := Part Ready;
END_TRANSITION
STEP CloseStopper1:
	CloseStopper1_action(N);
END_STEP
TRANSITION FROM CloseStopper1 TO CheckPos12full := State Ok;
END_TRANSITION
STEP CheckPos12full:
END_STEP
TRANSITION FROM CheckPos12full TO CheckCam2Active := Pos12Full;
END_TRANSITION
TRANSITION FROM CheckPos12full TO SeqEnd := TRUE;
END_TRANSITION
STEP CheckCam2Active:
	CheckCam2Active_action(N);
END_STEP
TRANSITION FROM CheckCam2Active TO Cam2_Start := Cam2Active;
END_TRANSITION
TRANSITION FROM CheckCam2Active TO Cam2_ResultOK := NotActive;
END_TRANSITION
STEP Cam2_Start:
	Cam2_Start_entry(P1);
	Cam2_Start_action(N);
END_STEP
TRANSITION FROM Cam2_Start TO Cam2_WaitDone := Busy;
END_TRANSITION
STEP Cam2_WaitDone:
	Cam2_WaitDone_entry(P1);
END_STEP
TRANSITION FROM Cam2_WaitDone TO Cam2_Result := Done;
END_TRANSITION
STEP Cam2_Result:
	Cam2_Result_action(N);
END_STEP
TRANSITION FROM Cam2_Result TO Cam2_Result_Counter := result_ok;
END_TRANSITION
TRANSITION FROM Cam2_Result TO Cam2_WaitRepeat := Repeat_;
END_TRANSITION
STEP Cam2_Result_Counter:
	Cam2_Result_Counter_entry(P1);
END_STEP
TRANSITION FROM Cam2_Result_Counter TO Result_Total := Cam2_CounterOK;
END_TRANSITION
TRANSITION FROM Cam2_Result_Counter TO Msg_Cam2 := Cam2_Nok;
END_TRANSITION
STEP Msg_Cam2:
	Msg_Cam2_entry(P1);
	Msg_Cam2_action(N);
	Msg_Cam2_exit(P0);
END_STEP
TRANSITION FROM Msg_Cam2 TO Cam2_CounterReset := MsgOK;
END_TRANSITION
TRANSITION FROM Msg_Cam2 TO CheckCam2Active := MsgCancel;
END_TRANSITION
STEP Cam2_CounterReset:
	Cam2_CounterReset_entry(P1);
END_STEP
TRANSITION FROM Cam2_CounterReset TO Result_Total := TRUE;
END_TRANSITION
STEP Cam2_WaitRepeat:
	Cam2_WaitRepeat_entry(P1);
	Cam2_WaitRepeat_action(N);
END_STEP
TRANSITION FROM Cam2_WaitRepeat TO Cam2_Start := Done;
END_TRANSITION
STEP Cam2_ResultOK:
	Cam2_ResultOK_entry(P1);
END_STEP
TRANSITION FROM Cam2_ResultOK TO Result_Total := TRUE;
END_TRANSITION
STEP Result_Total:
	Result_Total_entry(P1);
END_STEP
TRANSITION FROM Result_Total TO ResetLock := TRUE;
END_TRANSITION
STEP ResetLock:
	ResetLock_entry(P1);
END_STEP
TRANSITION FROM ResetLock TO SeqEnd := Tippbetrieb;
END_TRANSITION
STEP SeqEnd: (* -> WAIT *)
	SeqEnd_action(N);
END_STEP
TRANSITION FROM SeqEnd TO WaitForStart := TRUE;
END_TRANSITION

ACTION Init_action:
Start:=FALSE;
State:=STATE_WAIT;
MsgOK:=FALSE;
MsgCancel:=FALSE;
SFCRun:=FALSE;
Result:=RESULT_NON;
LockForCam:=FALSE;
END_ACTION

ACTION WaitForStart_action:
IF 	Start   THEN
	State:=STATE_RUN;
	SFCTimeStart:=TIME();
	Start:=FALSE;
ELSE
	State:=STATE_WAIT;
	MsgOK:=FALSE;
	MsgCancel:=FALSE;
	SFCRun:=FALSE;
END_IF
END_ACTION

ACTION Kamera_nicht_bb_entry:
MessageHandler.ClearMessageLines(sVisu:=Visu.Message);
END_ACTION

ACTION Kamera_nicht_bb_action:
(* Sensopart Kamera *)
IF	ST03_8_100_A1.Activated AND
	ST03_8_100_A1.sm_kamera_nicht_bb THEN
	MessageHandler.Msg.ID:='PM152';
	MessageHandler.Msg.Text:='Sesopart Kamera ist nicht betriebsbereit';

(* Keyence Kamera *)
ELSIF
	ST03_8_105_A1.sConfig.Aktiv AND
	ST03_8_105_A1.sm_kamera_nicht_bb THEN
	MessageHandler.Msg.ID:='PM159';
	MessageHandler.Msg.Text:='Keyence Kamera ist nicht betriebsbereit';
END_IF

	MessageHandler.Msg.Name:='Check Camera';
	MessageHandler.Msg.Color:=Color.red;
	MessageHandler.Msg.Station:=1;

	MessageHandler(
		Prio:=2, 							(*1=highest, .. , 4=lowest*)
		Btn1Addr:=ADR(MsgOk),			(*Address of Button1 , if Zero then Button is unvisible*)
		Btn2Addr:=,						(*Address of Button2 , if Zero then Button is unvisible*)
		sVisu:=Visu.Message);
END_ACTION

ACTION Kamera_nicht_bb_exit:
MsgOk:=FALSE;
MsgCancel:=FALSE;

(* Sensopart Kamera *)
IF ST03_8_100_A1.Activated THEN
	ST03_8_100_A1.st_ctrl_in.b_quitt := TRUE;
END_IF

(* Keyence Kamera *)
IF ST03_8_105_A1.sConfig.Aktiv THEN
	ST03_8_105_A1.st_ctrl_in.b_quitt := TRUE;
END_IF
END_ACTION

ACTION Wait_Reconnect_entry:
Delay(IN:=FALSE);
END_ACTION

ACTION Wait_Reconnect_action:
Delay(	IN:=TRUE, 		(*warte kurz, um neu zu verbinden *)
		PT:=T#1s);
END_ACTION

ACTION OpenSeperator_action:
ST03_4x3_Y70_5.MoveInit:=TRUE;		(*Zuführung Vereinzler AST/GST *)
END_ACTION

ACTION WaitForPart_entry:
ProcessMessage02:='';
Delay(IN:=FALSE);
END_ACTION

ACTION WaitForPart_action:
ProcessMessage02:='2IM6';				(*warte auf Teil Übergabeposition 1*)
Delay(	IN:=ST03_4x2_B69_5.BitInToCheck, (*ISK anwesend am Stopper*)
		PT:=T#50ms);
END_ACTION

ACTION WaitForPart_exit:
ProcessMessage02:='';
END_ACTION

ACTION CloseSeperator_action:
ST03_4x3_Y70_5.MoveWork:=TRUE;		(*Zuführung Vereinzler AST/GST *)
END_ACTION

ACTION OpenStopper_action:
ST03_4x3_Y70_6.MoveWork:=TRUE;		(*Zuführung Stopper AST/GST *)
END_ACTION

ACTION WaitForPartOnPos1_entry:
ProcessMessage02:='';
Delay(IN:=FALSE);
END_ACTION

ACTION WaitForPartOnPos1_action:
ProcessMessage02:='2IM6';					(*warte auf Teil Übergabeposition 1*)
Delay.IN:=ST03_4x3_B70_0.BitInToCheck;  	(*ISK anwesend Übergabeposition Stopper *)

Delay.PT:=T#50ms;
Delay();
END_ACTION

ACTION WaitForPartOnPos1_exit:
ProcessMessage02:='';
END_ACTION

ACTION CloseStopper_action:
ST03_4x3_Y70_6.MoveInit:=TRUE;		(*Zuführung Stopper AST/GST *)
END_ACTION

ACTION OpenSeperator__action:
ST03_4x3_Y70_5.MoveInit:=TRUE;		(*Zuführung Vereinzler AST/GST *)
END_ACTION

ACTION CheckCam1Active_action:
RepeatCounter:=0;

(* Teil 1 oder Teil 2*)
IF 	NOT ST03_4x3_B70_1.BitInToCheck AND		(* Teil vor Stopper bzw. Übergabeposition 1*)
	ST03_4x3_B70_0.BitInToCheck THEN		(* Teil nach Stopper bzw. Übergabeposition 2*)
	Part := 1;
ELSE
	Part := 2;
END_IF

LockForCam:=TRUE;
END_ACTION

ACTION Cam1_Start_entry:
Result_Cam1[Part] := RESULT_NON;
END_ACTION

ACTION Cam1_Start_action:
ST03_8_105_A1.JobNo := TD.Keyence_CamProgNo ;		(* Keyence Kameraprogramm*)
ST03_8_105_A1.st_ctrl_in.b_start := TRUE;
END_ACTION

ACTION Cam1_WaitDone_action:
ST03_8_105_A1.st_ctrl_in.b_start := FALSE;
RepeatCounter:=RepeatCounter+1;
END_ACTION

ACTION Cam1_Result_action:
IF 	(ST03_8_105_A1.b_Kam_Pruef_IO AND			 (*Kamera 1 = Keyence IV4*)
	NOT ST03_8_105_A1.b_Kam_Pruef_NIO) OR
	KeyenceCam_AlwaysOK THEN
	Result_Cam1[Part] := RESULT_OK;
ELSE
	Result_Cam1[Part] := RESULT_NOK;
END_IF
END_ACTION

ACTION Cam1_WaitRepeat_entry:
Delay(IN:=FALSE);
END_ACTION

ACTION Cam1_WaitRepeat_action:
Delay(	IN:=TRUE, 		(*warte kurz, bevor neues Bild gemacht wird *)
		PT:=T#500ms);
END_ACTION

ACTION Cam1_Result_Counter_entry:
FOR i:=100 TO 2 BY-1 DO
   NokPercent_Cam[1,i] := NokPercent_Cam[1,i-1];
END_FOR

IF 	Result_Cam1[Part] = RESULT_NOK THEN
	NokCounter_Cam[1] := NokCounter_Cam[1] + 1;
	NokPercent_Cam[1,1] := TRUE;
ELSE
	NokCounter_Cam[1] := 0;
	NokPercent_Cam[1,1] := FALSE;
END_IF

(*Anzahl der Schlechtteile von den letzten 100 Prüfungen*)
NokCounterPercent_Cam[1] := 0;
FOR i:=1 TO 100 BY 1 DO
	IF NokPercent_Cam[1,i] THEN
	NokCounterPercent_Cam[1] := NokCounterPercent_Cam[1]+1;
	END_IF
END_FOR
END_ACTION

ACTION Msg_Cam1_entry:
MessageHandler.ClearMessageLines(sVisu:=Visu.Message);
END_ACTION

ACTION Msg_Cam1_action:
IF NokCounter_Cam[1] >= MP.ST03.CamNoOfErrors_KYE THEN
	MessageHandler.Msg.ID:='PM124';
	MessageHandler.Msg.Name:='Keyence Kam.-Erg. Prüfung  n.i.o:';
	MessageHandler.Msg.Text:='Keyence Kam.-Erg. Prüfung  n.i.o: Fehler in Folge';

ELSIF NokCounterPercent_Cam[1] >= MP.ST03.CamNoOfErrorsPercent_KYE THEN
	MessageHandler.Msg.ID:='PM125';
	MessageHandler.Msg.Name:='Keyence Kam.-Erg. Prüfung  n.i.o:';
	MessageHandler.Msg.Text:='Keyence Kam.-Erg. Prüfung  n.i.o:% Fehler';

END_IF

	MessageHandler.Msg.Color:=Color.red;
	MessageHandler.Msg.Station:=3;
	MessageHandler.MsgButton1Text:='continue';
	MessageHandler.MsgButton2Text:='repeat';
	
	MessageHandler(
		Prio:=2, 								(*1=highest, .. , 4=lowest*)
		Btn1Addr:=ADR(MsgOk),				(*Address of Button1 , if Zero then Button is unvisible*)
		Btn2Addr:=ADR(MsgCancel),			(*Address of Button2 , if Zero then Button is unvisible*)
		sVisu:=Visu.Message);
END_ACTION

ACTION Msg_Cam1_exit:
MsgOk:=FALSE;
MsgCancel:=FALSE;
END_ACTION

ACTION Cam1_CounterReset_entry:
NokCounter_Cam[1] := 0;
NokCounterPercent_Cam[1] := 0;
(*Percent Register löschen*)
FOR i:=1 TO 100 BY 1 DO
  NokPercent_Cam[1,i]:= FALSE;
END_FOR
END_ACTION

ACTION ResultCam1OK_action:
Result_Cam1[1] := RESULT_OK;
Result_Cam1[2] := RESULT_OK;
END_ACTION

ACTION OpenStopper1__action:
ST03_4x3_Y70_7.MoveWork:=TRUE;		(* Zuführung Stopper Übergabeposition AST/GST*)
END_ACTION

ACTION WaitForPartOnPos2_entry:
ProcessMessage02:='';
Delay(IN:=FALSE);
END_ACTION

ACTION WaitForPartOnPos2_action:
ProcessMessage02:='2IM5';						(*warte auf Teil Übergabeposition 2*)
Delay(	IN:=ST03_4x3_B70_1.BitInToCheck, 		(*ISK anwesend Übergabeposition *)
		PT:=T#50ms);
END_ACTION

ACTION WaitForPartOnPos2_exit:
ProcessMessage02:='';
END_ACTION

ACTION CloseStopper1_action:
ST03_4x3_Y70_7.MoveInit:=TRUE;		(* Zuführung Stopper Übergabeposition AST/GST *)
END_ACTION

ACTION CheckCam2Active_action:
RepeatCounter:=0;
END_ACTION

ACTION Cam2_Start_entry:
Result_Cam2 := RESULT_NON;
END_ACTION

ACTION Cam2_Start_action:
ST03_8_100_A1.JobNo := TD.Sensopart_CamProgNo ;
ST03_8_100_A1.st_ctrl_in.b_start := TRUE;
END_ACTION

ACTION Cam2_WaitDone_entry:
ST03_8_100_A1.st_ctrl_in.b_start := FALSE;
RepeatCounter:=RepeatCounter+1;
END_ACTION

ACTION Cam2_Result_action:
IF 	(ST03_8_100_A1.b_Kam_Pruef_IO AND			 (*Kamera 2 = Sensopart V20*)
	NOT ST03_8_100_A1.b_Kam_Pruef_NIO) OR
	SensopartCam_AlwaysOK THEN
	Result_Cam2 := RESULT_OK;
ELSE
	Result_Cam2 := RESULT_NOK;
END_IF
END_ACTION

ACTION Cam2_Result_Counter_entry:
FOR i:=100 TO 2 BY-1 DO
   NokPercent_Cam[2,i] := NokPercent_Cam[2,i-1];
END_FOR

IF	Result_Cam2 = RESULT_OK THEN
	NokCounter_Cam[2] := 0;
	NokPercent_Cam[2,1] := FALSE;
ELSE
	NokCounter_Cam[2] := NokCounter_Cam[2] + 1;
	NokPercent_Cam[2,1] := TRUE;
END_IF

(*Anzahl der Schlechtteile von den letzten 100 Prüfungen*)
NokCounterPercent_Cam[2] := 0;
FOR i:=1 TO 100 BY 1 DO
	IF NokPercent_Cam[2,i] THEN
	NokCounterPercent_Cam[2] := NokCounterPercent_Cam[2]+1;
	END_IF
END_FOR
END_ACTION

ACTION Msg_Cam2_entry:
MessageHandler.ClearMessageLines(sVisu:=Visu.Message);
END_ACTION

ACTION Msg_Cam2_action:
IF NokCounter_Cam[2] >= MP.ST03.CamNoOfErrors THEN
	MessageHandler.Msg.ID:='PM112';
	MessageHandler.Msg.Name:='Sensopart Kam.-Erg. Prüfung  n.i.o:';
	MessageHandler.Msg.Text:='Sensopart Kam.-Erg. Prüfung  n.i.o: Fehler in Folge';

ELSIF NokCounterPercent_Cam[2] >= MP.ST03.CamNoOfErrorsPercent THEN
	MessageHandler.Msg.ID:='PM113';
	MessageHandler.Msg.Name:='Sensopart Kam.-Erg. Prüfung  n.i.o:';
	MessageHandler.Msg.Text:='Sensopart Kam.-Erg. Prüfung  n.i.o:% Fehler';
END_IF

	MessageHandler.Msg.Color:=Color.red;
	MessageHandler.Msg.Station:=3;
	MessageHandler.MsgButton1Text:='continue';
	MessageHandler.MsgButton2Text:='repeat';
	
	MessageHandler(
		Prio:=2, 								(*1=highest, .. , 4=lowest*)
		Btn1Addr:=ADR(MsgOk),				(*Address of Button1 , if Zero then Button is unvisible*)
		Btn2Addr:=ADR(MsgCancel),			(*Address of Button2 , if Zero then Button is unvisible*)
		sVisu:=Visu.Message);
END_ACTION

ACTION Msg_Cam2_exit:
MsgOk:=FALSE;
MsgCancel:=FALSE;
END_ACTION

ACTION Cam2_CounterReset_entry:
NokCounter_Cam[2] := 0;
NokCounterPercent_Cam[2] := 0;
(*Percent Register löschen*)
FOR i:=1 TO 100 BY 1 DO
  NokPercent_Cam[2,i]:= FALSE;
END_FOR
END_ACTION

ACTION Cam2_WaitRepeat_entry:
Delay(IN:=FALSE);
END_ACTION

ACTION Cam2_WaitRepeat_action:
Delay(	IN:=TRUE, 		(*warte kurz, bevor neues Bild gemacht wird *)
		PT:=T#750ms);
END_ACTION

ACTION Cam2_ResultOK_entry:
Result_Cam2 := RESULT_OK;
END_ACTION

ACTION Result_Total_entry:
IF	Result_Cam1[1] = RESULT_OK AND
	Result_Cam1[2] = RESULT_OK AND
	Result_Cam2 = RESULT_OK THEN
	Result := RESULT_OK;
ELSE
	Result := RESULT_NOK;
	gNokPartsColorCam := gNokPartsColorCam + 1;
END_IF
END_ACTION

ACTION ResetLock_entry:
LockForCam:=FALSE;
END_ACTION

ACTION SeqEnd_action:
SFCTime:=TIME_TO_DINT(TIME()-SFCTimeStart);
State:=STATE_WAIT;
END_ACTION

TRANSITION Kamera_betriebsbereit:
(*Kamera betriebsbereit oder nicht Aktiv*)

(* Sensopart Kamera *)
(NOT ST03_8_100_A1.Activated OR
ST03_8_100_A1.Activated AND
NOT ST03_8_100_A1.sm_kamera_nicht_bb) AND
(* Keyence Kamera *)
(NOT ST03_8_105_A1.sConfig.Aktiv OR
ST03_8_105_A1.sConfig.Aktiv AND
NOT ST03_8_105_A1.sm_kamera_nicht_bb)
END_TRANSITION

TRANSITION Done:
Delay.Q
END_TRANSITION

TRANSITION Check_Part:
Robot01.ActualArea <> 4 AND (
NOT ST03_4x3_B70_0.BitInToCheck OR	(* ISK anwesend Übergabeposition Stopper*)
NOT ST03_4x3_B70_1.BitInToCheck )	(* ISK anwesend Übergabeposition*)
END_TRANSITION

TRANSITION PosEmpty:
NOT ST03_4x2_B69_5.BitInToCheck			 	(*  ISK anwesend am Stopper*)
END_TRANSITION

TRANSITION State Ok:
ST03_4x3_Y70_5.State=STATE_OK (*Zuführung Vereinzler AST/GST *)
END_TRANSITION

TRANSITION Part Ready:
Delay.Q
END_TRANSITION

TRANSITION PosFull:
ST03_4x2_B69_5.BitInToCheck			 	(*  ISK anwesend am Stopper*)
END_TRANSITION

TRANSITION State Ok:
ST03_4x3_Y70_5.State=STATE_OK (*Zuführung Vereinzler AST/GST *)
END_TRANSITION

TRANSITION Pos1Empty:
NOT ST03_4x3_B70_0.BitInToCheck AND 	(*  ISK anwesend Übergabeposition Stopper*)
ST03_4x2_B69_5.BitInToCheck			 	(*  ISK anwesend am Stopper*)
END_TRANSITION

TRANSITION State Ok:
ST03_4x3_Y70_6.State=STATE_OK 	(*Zuführung Stopper AST/GST *)
END_TRANSITION

TRANSITION Pos2Empty:
ST03_4x3_B70_0.BitInToCheck AND 	(*  ISK anwesend Übergabeposition Stopper*)
NOT ST03_4x3_B70_1.BitInToCheck AND 	(*  ISK anwesend Übergabeposition*)
ST03_4x2_B69_5.BitInToCheck			 	(*  ISK anwesend am Stopper*)
END_TRANSITION

TRANSITION Part Ready:
Delay.Q
END_TRANSITION

TRANSITION Pos1Full:
ST03_4x3_B70_0.BitInToCheck 	(*ISK anwesend Übergabeposition Stopper*)
END_TRANSITION

TRANSITION State Ok:
ST03_4x3_Y70_6.State=STATE_OK AND	(*Zuführung Stopper AST/GST *)
ST03_4x3_Y70_5.State=STATE_OK (*Zuführung Vereinzler AST/GST *)
END_TRANSITION

TRANSITION Cam1Active:
ST03_8_105_A1.sConfig.Aktiv
END_TRANSITION

TRANSITION Busy:
ST03_8_105_A1.st_ctrl_out.b_busy	 (*Kamera Ehternet*)
END_TRANSITION

TRANSITION Done:
ST03_8_105_A1.st_ctrl_out.b_fertig
END_TRANSITION

TRANSITION result_ok:
Result_Cam1[Part] = RESULT_OK OR
RepeatCounter >= 2
END_TRANSITION

TRANSITION Repeat_:
TRUE
END_TRANSITION

TRANSITION Done:
Delay.Q
END_TRANSITION

TRANSITION Cam1_CounterOK:
NokCounter_Cam[1] < MP.ST03.CamNoOfErrors_KYE AND
NokCounterPercent_Cam[1] < MP.ST03.CamNoOfErrorsPercent_KYE
END_TRANSITION

TRANSITION Cam1_Nok:
NokCounter_Cam[1] >= MP.ST03.CamNoOfErrors_KYE OR
NokCounterPercent_Cam[1] >= MP.ST03.CamNoOfErrorsPercent_KYE
END_TRANSITION

TRANSITION NotActive:
TRUE
END_TRANSITION

TRANSITION Tippbetrieb:
gTipImp
END_TRANSITION

TRANSITION Pos2Empty:
NOT ST03_4x3_B70_1.BitInToCheck AND 	(*  ISK anwesend Übergabeposition*)
ST03_4x3_B70_0.BitInToCheck			 	(*  ISK anwesend Übergabeposition Stopper*)
END_TRANSITION

TRANSITION State Ok:
ST03_4x3_Y70_7.State=STATE_OK 	(* Zuführung Stopper Übergabeposition AST/GST *)
END_TRANSITION

TRANSITION Part Ready:
Delay.Q
END_TRANSITION

TRANSITION Pos2Full:
ST03_4x3_B70_1.BitInToCheck	 	(*ISK anwesend Übergabeposition*)
END_TRANSITION

TRANSITION State Ok:
ST03_4x3_Y70_7.State=STATE_OK 	(* Zuführung Stopper Übergabeposition AST/GST *)
END_TRANSITION

TRANSITION Pos12Full:
ST03_4x3_B70_0.BitInToCheck AND		(*  ISK anwesend Übergabeposition 1*)
ST03_4x3_B70_1.BitInToCheck		 	(*  ISK anwesend Übergabeposition 2*)
END_TRANSITION

TRANSITION Cam2Active:
ST03_8_100_A1.Activated
END_TRANSITION

TRANSITION Busy:
ST03_8_100_A1.st_ctrl_out.b_busy 	(*Kamera Farberkennung Ehternet*)
END_TRANSITION

TRANSITION Done:
ST03_8_100_A1.st_ctrl_out.b_fertig
END_TRANSITION

TRANSITION result_ok:
Result_Cam2 = RESULT_OK OR
RepeatCounter >= 2
END_TRANSITION

TRANSITION Cam2_CounterOK:
NokCounter_Cam[2] < MP.ST03.CamNoOfErrors AND
NokCounterPercent_Cam[2] < MP.ST03.CamNoOfErrorsPercent
END_TRANSITION

TRANSITION Cam2_Nok:
NokCounter_Cam[2] >= MP.ST03.CamNoOfErrors OR
NokCounterPercent_Cam[2] >= MP.ST03.CamNoOfErrorsPercent
END_TRANSITION

TRANSITION Repeat_:
TRUE
END_TRANSITION

TRANSITION Done:
Delay.Q
END_TRANSITION

TRANSITION NotActive:
TRUE
END_TRANSITION

TRANSITION Tippbetrieb:
gTipImp
END_TRANSITION
END_PROGRAM

(* POU Stations/ST_00/ST00_SFCs/_SpecialModeSFCs/CallSpecialModeSFCs, ST *)
PROGRAM CallSpecialModeSFCs
VAR_OUTPUT
  AllSpecialModeSFCInInit : BOOL := TRUE;

END_VAR
SpecialModeMain();
SpecialMode01();
SpecialMode02();
SpecialMode03();
SpecialMode04();
SpecialMode05();
SpecialMode06();
SpecialMode07();
SpecialMode08();

AllSpecialModeSFCInInit:=SpecialModeMain.State=STATE_OK;
END_PROGRAM

(* POU Stations/ST_00/ST00_SFCs/_SpecialModeSFCs/SpecialModeMain, SFC *)
PROGRAM SpecialModeMain
(* 09.MAY 2005 Ext/g.baiz *)

VAR_OUTPUT
	SFCCurrentPOU		: STRING:='SpecialModeMain';
	SFCCurrentStep	: STRING:='';
	SFCTime					:	DINT;
  State   				:	DINT;
  Result  				:	DINT;
END_VAR
VAR_INPUT
	ModeNo					: DINT;
END_VAR
VAR
	MsgOK				:	BOOL;
	MsgCancel		:	BOOL;
	SFCRun					:	BOOL;
	SFCTimeStart		:	TIME;
	(* Userdefinded area *)
	SpecMode01Flag	:	R_TRIG;
	SpecMode02Flag	:	R_TRIG;
	SpecMode03Flag	:	R_TRIG;
	SpecMode04Flag	:	R_TRIG;
	SpecMode05Flag	:	R_TRIG;
	SpecMode06Flag	:	R_TRIG;
	SpecMode07Flag	:	R_TRIG;
	SpecMode08Flag	:	R_TRIG;

	idx							:	INT;

END_VAR
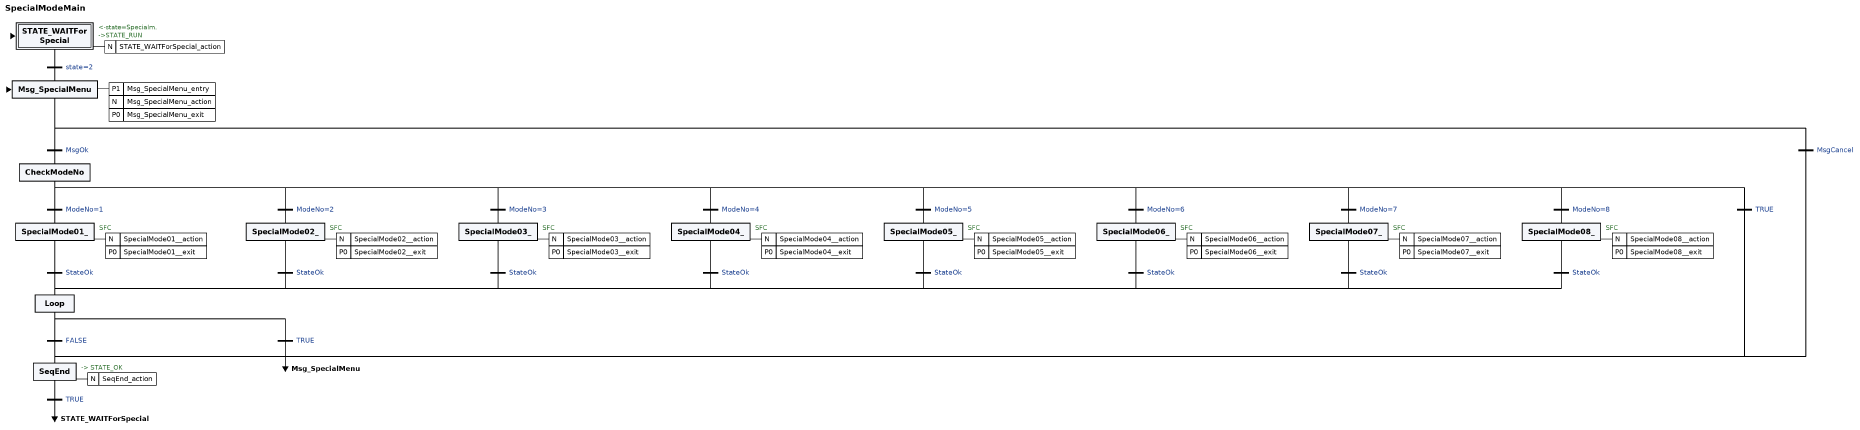
INITIAL_STEP STATE_WAITForSpecial: (* <-state=Specialm. / ->STATE_RUN *)
	STATE_WAITForSpecial_action(N);
END_STEP
TRANSITION FROM STATE_WAITForSpecial TO Msg_SpecialMenu := state=2;
END_TRANSITION
STEP Msg_SpecialMenu:
	Msg_SpecialMenu_entry(P1);
	Msg_SpecialMenu_action(N);
	Msg_SpecialMenu_exit(P0);
END_STEP
TRANSITION FROM Msg_SpecialMenu TO CheckModeNo := MsgOk;
END_TRANSITION
TRANSITION FROM Msg_SpecialMenu TO SeqEnd := MsgCancel;
END_TRANSITION
STEP CheckModeNo:
END_STEP
TRANSITION FROM CheckModeNo TO SpecialMode01_ := ModeNo=1;
END_TRANSITION
TRANSITION FROM CheckModeNo TO SpecialMode02_ := ModeNo=2;
END_TRANSITION
TRANSITION FROM CheckModeNo TO SpecialMode03_ := ModeNo=3;
END_TRANSITION
TRANSITION FROM CheckModeNo TO SpecialMode04_ := ModeNo=4;
END_TRANSITION
TRANSITION FROM CheckModeNo TO SpecialMode05_ := ModeNo=5;
END_TRANSITION
TRANSITION FROM CheckModeNo TO SpecialMode06_ := ModeNo=6;
END_TRANSITION
TRANSITION FROM CheckModeNo TO SpecialMode07_ := ModeNo=7;
END_TRANSITION
TRANSITION FROM CheckModeNo TO SpecialMode08_ := ModeNo=8;
END_TRANSITION
TRANSITION FROM CheckModeNo TO SeqEnd := TRUE;
END_TRANSITION
STEP SpecialMode01_: (* SFC *)
	SpecialMode01__action(N);
	SpecialMode01__exit(P0);
END_STEP
TRANSITION FROM SpecialMode01_ TO Loop := StateOk;
END_TRANSITION
STEP SpecialMode02_: (* SFC *)
	SpecialMode02__action(N);
	SpecialMode02__exit(P0);
END_STEP
TRANSITION FROM SpecialMode02_ TO Loop := StateOk;
END_TRANSITION
STEP SpecialMode03_: (* SFC *)
	SpecialMode03__action(N);
	SpecialMode03__exit(P0);
END_STEP
TRANSITION FROM SpecialMode03_ TO Loop := StateOk;
END_TRANSITION
STEP SpecialMode04_: (* SFC *)
	SpecialMode04__action(N);
	SpecialMode04__exit(P0);
END_STEP
TRANSITION FROM SpecialMode04_ TO Loop := StateOk;
END_TRANSITION
STEP SpecialMode05_: (* SFC *)
	SpecialMode05__action(N);
	SpecialMode05__exit(P0);
END_STEP
TRANSITION FROM SpecialMode05_ TO Loop := StateOk;
END_TRANSITION
STEP SpecialMode06_: (* SFC *)
	SpecialMode06__action(N);
	SpecialMode06__exit(P0);
END_STEP
TRANSITION FROM SpecialMode06_ TO Loop := StateOk;
END_TRANSITION
STEP SpecialMode07_: (* SFC *)
	SpecialMode07__action(N);
	SpecialMode07__exit(P0);
END_STEP
TRANSITION FROM SpecialMode07_ TO Loop := StateOk;
END_TRANSITION
STEP SpecialMode08_: (* SFC *)
	SpecialMode08__action(N);
	SpecialMode08__exit(P0);
END_STEP
TRANSITION FROM SpecialMode08_ TO Loop := StateOk;
END_TRANSITION
STEP Loop:
END_STEP
TRANSITION FROM Loop TO SeqEnd := FALSE;
END_TRANSITION
TRANSITION FROM Loop TO Msg_SpecialMenu := TRUE;
END_TRANSITION
STEP SeqEnd: (* -> STATE_OK *)
	SeqEnd_action(N);
END_STEP
TRANSITION FROM SeqEnd TO STATE_WAITForSpecial := TRUE;
END_TRANSITION

ACTION STATE_WAITForSpecial_action:
IF 	ModeSelect.Mode=MODE_SPECIAL
THEN
	State:=STATE_RUN;
	Result:=RESULT_NON;
	SFCTimeStart:=TIME();
ELSE
	State:=STATE_WAIT;
	SFCRun:=FALSE;
END_IF
END_ACTION

ACTION Msg_SpecialMenu_entry:
MessageHandler.ClearMessageLines(sVisu:=Visu.Message);

idx:=1;
MessageHandler.MessageLine[idx].Visible:=FALSE;
MessageHandler.MessageLine[idx].Editable:=TRUE;
MessageHandler.MessageLine[idx].Text:='Specialmode_1';				(*Ablauf Pallettierer*)
MessageHandler.MessageLine[idx].MsgInt:=1;
MessageHandler.MessageLine[idx].MsgBool:=FALSE;
MessageHandler.MessageLine[idx].MsgTypeEnum:=MsgDataTypeBool;

idx:=idx+1;
MessageHandler.MessageLine[idx].Visible:=FALSE;
MessageHandler.MessageLine[idx].Editable:=TRUE;
MessageHandler.MessageLine[idx].Text:='Specialmode_2';				(*Not used*)
MessageHandler.MessageLine[idx].MsgInt:=2;
MessageHandler.MessageLine[idx].MsgBool:=FALSE;
MessageHandler.MessageLine[idx].MsgTypeEnum:=MsgDataTypeBool;

idx:=idx+1;
MessageHandler.MessageLine[idx].Visible:=FALSE;
MessageHandler.MessageLine[idx].Editable:=TRUE;
MessageHandler.MessageLine[idx].Text:='Specialmode_3';				(*Not used*)
MessageHandler.MessageLine[idx].MsgInt:=3;
MessageHandler.MessageLine[idx].MsgBool:=FALSE;
MessageHandler.MessageLine[idx].MsgTypeEnum:=MsgDataTypeBool;

idx:=idx+1;
MessageHandler.MessageLine[idx].Visible:=FALSE;
MessageHandler.MessageLine[idx].Editable:=TRUE;
MessageHandler.MessageLine[idx].Text:='Specialmode_4';				(*Not used*)
MessageHandler.MessageLine[idx].MsgInt:=4;
MessageHandler.MessageLine[idx].MsgBool:=FALSE;
MessageHandler.MessageLine[idx].MsgTypeEnum:=MsgDataTypeBool;

idx:=idx+1;
MessageHandler.MessageLine[idx].Visible:=FALSE;
MessageHandler.MessageLine[idx].Editable:=TRUE;
MessageHandler.MessageLine[idx].Text:='Specialmode_5';				(*Blister Abstapeln*)
MessageHandler.MessageLine[idx].MsgInt:=5;
MessageHandler.MessageLine[idx].MsgBool:=FALSE;
MessageHandler.MessageLine[idx].MsgTypeEnum:=MsgDataTypeBool;

idx:=idx+1;
MessageHandler.MessageLine[idx].Visible:=gTypeCode=312 OR gTypeCode=499 OR gTypeCode=322;	(*93pol*)(*102pol*)(*160pol*);
MessageHandler.MessageLine[idx].Editable:=TRUE;
MessageHandler.MessageLine[idx].Text:='Specialmode_6';				(*Dummytest*)
MessageHandler.MessageLine[idx].MsgInt:=6;
MessageHandler.MessageLine[idx].MsgBool:=FALSE;
MessageHandler.MessageLine[idx].MsgTypeEnum:=MsgDataTypeBool;

idx:=idx+1;
MessageHandler.MessageLine[idx].Visible:=FALSE;
MessageHandler.MessageLine[idx].Editable:=TRUE;
MessageHandler.MessageLine[idx].Text:='Specialmode_7';				(*Not used*)
MessageHandler.MessageLine[idx].MsgInt:=7;
MessageHandler.MessageLine[idx].MsgBool:=FALSE;
MessageHandler.MessageLine[idx].MsgTypeEnum:=MsgDataTypeBool;

idx:=idx+1;
MessageHandler.MessageLine[idx].Visible:=FALSE;
MessageHandler.MessageLine[idx].Editable:=TRUE;
MessageHandler.MessageLine[idx].Text:='Specialmode_8';				(*Not used*)
MessageHandler.MessageLine[idx].MsgInt:=8;
MessageHandler.MessageLine[idx].MsgBool:=FALSE;
MessageHandler.MessageLine[idx].MsgTypeEnum:=MsgDataTypeBool;

IF 	ModeNo>=1 AND
	ModeNo<=8 THEN
	MessageHandler.MessageLine[ModeNo].MsgBool:=TRUE;
END_IF
END_ACTION

ACTION Msg_SpecialMenu_action:
MessageHandler.Msg.ID:='PM61';
MessageHandler.Msg.Name:='Teil-Abläufe';
MessageHandler.Msg.Text:='Teilablauf auswählen und mit OK starten';
MessageHandler.Msg.Color:=Color.yellow;
MessageHandler.Msg.Station:=0;


MessageHandler(
	Prio:=2, 					(*1=highest, .. , 4=lowest*)
	Btn1Addr:=ADR(MsgOk),		(*Address of Button1 , if Zero then Button is unvisible*)
	Btn2Addr:=ADR(MsgCancel),	(*Address of Button2 , if Zero then Button is unvisible*)
	sVisu:=Visu.Message);

MessageHandler.DisableMultiSelect(sVisu:=Visu.Message);

FOR idx:=1 TO 10 DO
	IF 	MessageHandler.MessageLine[idx].MsgBool THEN
		ModeNo:=idx;
	END_IF
END_FOR
END_ACTION

ACTION Msg_SpecialMenu_exit:
MsgOk:=FALSE;
MsgCancel:=FALSE;
END_ACTION

ACTION SpecialMode01__action:
IF SpecialMode01.State=STATE_WAIT
THEN
	SpecialMode01(Start:=TRUE);

	SFCRun:=TRUE;
(*ELSE*)
END_IF
END_ACTION

ACTION SpecialMode01__exit:
SpecialMode01.Start:=FALSE;
SFCRun:=FALSE;
END_ACTION

ACTION SpecialMode02__action:
IF SpecialMode02.State=STATE_WAIT
THEN
	SpecialMode02(Start:=TRUE);

	SFCRun:=TRUE;
(*ELSE*)
END_IF
END_ACTION

ACTION SpecialMode02__exit:
SpecialMode02.Start:=FALSE;
SFCRun:=FALSE;
END_ACTION

ACTION SpecialMode03__action:
IF SpecialMode03.State=STATE_WAIT
THEN
	SpecialMode03(Start:=TRUE);

	SFCRun:=TRUE;
(*ELSE*)
END_IF
END_ACTION

ACTION SpecialMode03__exit:
SpecialMode03.Start:=FALSE;
SFCRun:=FALSE;
END_ACTION

ACTION SpecialMode04__action:
IF SpecialMode04.State=STATE_WAIT
THEN
	SpecialMode04(Start:=TRUE);

	SFCRun:=TRUE;
(*ELSE*)
END_IF
END_ACTION

ACTION SpecialMode04__exit:
SpecialMode04.Start:=FALSE;
SFCRun:=FALSE;
END_ACTION

ACTION SpecialMode05__action:
IF SpecialMode05.State=STATE_WAIT
THEN
	SpecialMode05(Start:=TRUE);

	SFCRun:=TRUE;
(*ELSE*)
END_IF
END_ACTION

ACTION SpecialMode05__exit:
SpecialMode05.Start:=FALSE;
SFCRun:=FALSE;
END_ACTION

ACTION SpecialMode06__action:
IF SpecialMode06.State=STATE_WAIT
THEN
	SpecialMode06(Start:=TRUE);

	IF	gTypeCode=312 OR		(*93pol*)
		gTypeCode=499 THEN		(*102pol*)
		MP.ST02.DummyPruefung_93pol  := TRUE;
	ELSIF
		gTypeCode=322	THEN	(*160pol*)
		DummyTest_160pol := TRUE;
	END_IF
	SFCRun:=TRUE;
END_IF
END_ACTION

ACTION SpecialMode06__exit:
SpecialMode06.Start:=FALSE;
SFCRun:=FALSE;
DummyTest_160pol := FALSE;
MP.ST02.DummyPruefung_93pol  := FALSE;
END_ACTION

ACTION SpecialMode07__action:
IF SpecialMode07.State=STATE_WAIT
THEN
	SpecialMode07(Start:=TRUE);

	SFCRun:=TRUE;
(*ELSE*)
END_IF
END_ACTION

ACTION SpecialMode07__exit:
SpecialMode07.Start:=FALSE;
SFCRun:=FALSE;
END_ACTION

ACTION SpecialMode08__action:
IF SpecialMode08.State=STATE_WAIT
THEN
	SpecialMode08(Start:=TRUE);

	SFCRun:=TRUE;
(*ELSE*)
END_IF
END_ACTION

ACTION SpecialMode08__exit:
SpecialMode08.Start:=FALSE;
SFCRun:=FALSE;
END_ACTION

ACTION SeqEnd_action:
SFCTime:=TIME_TO_DINT(TIME()-SFCTimeStart);
State:=STATE_OK;
END_ACTION

TRANSITION ModeNo=1:
ModeNo=1
END_TRANSITION

TRANSITION StateOk:
		SFCRun=TRUE
AND SpecialMode01.State=STATE_OK
END_TRANSITION

TRANSITION ModeNo=2:
ModeNo=2
END_TRANSITION

TRANSITION StateOk:
		SFCRun=TRUE
AND SpecialMode02.State=STATE_OK
END_TRANSITION

TRANSITION ModeNo=3:
ModeNo=3
END_TRANSITION

TRANSITION StateOk:
		SFCRun=TRUE
AND SpecialMode03.State=STATE_OK
END_TRANSITION

TRANSITION ModeNo=4:
ModeNo=4
END_TRANSITION

TRANSITION StateOk:
		SFCRun=TRUE
AND SpecialMode04.State=STATE_OK
END_TRANSITION

TRANSITION ModeNo=5:
ModeNo=5
END_TRANSITION

TRANSITION StateOk:
		SFCRun=TRUE
AND SpecialMode05.State=STATE_OK
END_TRANSITION

TRANSITION ModeNo=6:
ModeNo=6
END_TRANSITION

TRANSITION StateOk:
		SFCRun=TRUE
AND SpecialMode06.State=STATE_OK
END_TRANSITION

TRANSITION ModeNo=7:
ModeNo=7
END_TRANSITION

TRANSITION StateOk:
		SFCRun=TRUE
AND SpecialMode07.State=STATE_OK
END_TRANSITION

TRANSITION ModeNo=8:
ModeNo=8
END_TRANSITION

TRANSITION StateOk:
		SFCRun=TRUE
AND SpecialMode08.State=STATE_OK
END_TRANSITION
END_PROGRAM

(* POU Stations/ST_00/ST00_SFCs/_SpecialModeSFCs/SpecialMode02, SFC *)
PROGRAM SpecialMode02 (*Used for: Prozess Kamera *)
(* Date:     Author:   *)

VAR_OUTPUT
	SFCCurrentPOU		: STRING:='SpecialMode02';
	SFCCurrentStep	: STRING:='';
	SFCTime					:	DINT;
  State   				:	DINT;
  Result  				:	DINT;
END_VAR
VAR_INPUT
	Start						:	BOOL;
END_VAR
VAR
	MsgOK				:	BOOL;
	MsgCancel		:	BOOL;
	SFCRun					:	BOOL;
	SFCTimeStart		:	TIME;

	(* Userdefinded area *)


END_VAR
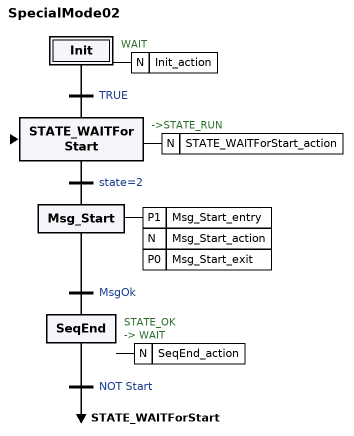
INITIAL_STEP Init: (* WAIT *)
	Init_action(N);
END_STEP
TRANSITION FROM Init TO STATE_WAITForStart := TRUE;
END_TRANSITION
STEP STATE_WAITForStart: (* ->STATE_RUN *)
	STATE_WAITForStart_action(N);
END_STEP
TRANSITION FROM STATE_WAITForStart TO Msg_Start := state=2;
END_TRANSITION
STEP Msg_Start:
	Msg_Start_entry(P1);
	Msg_Start_action(N);
	Msg_Start_exit(P0);
END_STEP
TRANSITION FROM Msg_Start TO SeqEnd := MsgOk;
END_TRANSITION
STEP SeqEnd: (* STATE_OK / -> WAIT *)
	SeqEnd_action(N);
END_STEP
TRANSITION FROM SeqEnd TO STATE_WAITForStart := NOT Start;
END_TRANSITION

ACTION Init_action:
Start:=FALSE;
State:=STATE_WAIT;
END_ACTION

ACTION STATE_WAITForStart_action:
IF Start=TRUE
THEN
	State:=STATE_RUN;
	Result:=RESULT_NON;
	SFCTimeStart:=TIME();
(*ELSE*)
END_IF
END_ACTION

ACTION Msg_Start_entry:
MessageHandler.ClearMessageLines(sVisu:=Visu.Message);
END_ACTION

ACTION Msg_Start_action:
MessageHandler.Msg.ID:='PM51';
MessageHandler.Msg.Name:='SpecialMode02_Start';
MessageHandler.Msg.Text:='Special Mode 2';
MessageHandler.Msg.Color:=Color.yellow;
MessageHandler.Msg.Station:=1;


MessageHandler(
	Prio:=2, 									(*1=highest, .. , 4=lowest*)
	Btn1Addr:=ADR(MsgOk),			(*Address of Button1 , if Zero then Button is unvisible*)
	Btn2Addr:=ADR(MsgCancel),	(*Address of Button2 , if Zero then Button is unvisible*)
	sVisu:=Visu.Message);


MessageHandler.MessageLine[1].Visible:=TRUE;
MessageHandler.MessageLine[1].Editable:=TRUE;
MessageHandler.MessageLine[1].Text:='Kamera Programm ';
MessageHandler.MessageLine[1].MsgTypeEnum:=MsgDataTypeDint;
END_ACTION

ACTION Msg_Start_exit:
MsgOk:=FALSE;
MsgCancel:=FALSE;
SpecialModeProgNu:=MessageHandler.MessageLine[1].MsgInt;
END_ACTION

ACTION SeqEnd_action:
IF 	State=STATE_RUN THEN
	SFCTime:=TIME_TO_DINT(TIME()-SFCTimeStart);
	State:=STATE_OK;
END_IF

IF 	NOT Start THEN
	State:=STATE_WAIT;
END_IF
END_ACTION
END_PROGRAM

(* POU Stations/ST_00/ST00_SFCs/_SpecialModeSFCs/SpecialMode04, SFC *)
PROGRAM SpecialMode04 (*not used*)
(* Date:     Author:   *)

VAR_OUTPUT
	SFCCurrentPOU		: STRING:='SpecialMode04';
	SFCCurrentStep		: STRING:='';
	SFCTime				: DINT;
	State   			: DINT;
	Result  			: DINT;
END_VAR
VAR_INPUT
	Start				: BOOL;
END_VAR
VAR
	MsgOK				: BOOL;
	MsgCancel			: BOOL;
	SFCRun				: BOOL;
	SFCTimeStart		: TIME;
	ResultString		: STRING;
	(* Userdefinded area *)



END_VAR
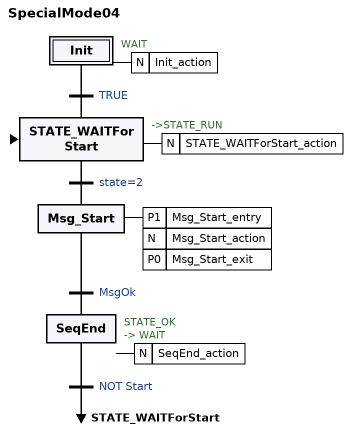
INITIAL_STEP Init: (* WAIT *)
	Init_action(N);
END_STEP
TRANSITION FROM Init TO STATE_WAITForStart := TRUE;
END_TRANSITION
STEP STATE_WAITForStart: (* ->STATE_RUN *)
	STATE_WAITForStart_action(N);
END_STEP
TRANSITION FROM STATE_WAITForStart TO Msg_Start := state=2;
END_TRANSITION
STEP Msg_Start:
	Msg_Start_entry(P1);
	Msg_Start_action(N);
	Msg_Start_exit(P0);
END_STEP
TRANSITION FROM Msg_Start TO SeqEnd := MsgOk;
END_TRANSITION
STEP SeqEnd: (* STATE_OK / -> WAIT *)
	SeqEnd_action(N);
END_STEP
TRANSITION FROM SeqEnd TO STATE_WAITForStart := NOT Start;
END_TRANSITION

ACTION Init_action:
Start:=FALSE;
State:=STATE_WAIT;
END_ACTION

ACTION STATE_WAITForStart_action:
IF Start=TRUE
THEN
	State:=STATE_RUN;
	Result:=RESULT_NON;
	SFCTimeStart:=TIME();
(*ELSE*)
END_IF
END_ACTION

ACTION Msg_Start_entry:
MessageHandler.ClearMessageLines(sVisu:=Visu.Message);
END_ACTION

ACTION Msg_Start_action:
MessageHandler.Msg.ID:='PM52';
MessageHandler.Msg.Name:='SpecialMode04_Start';
MessageHandler.Msg.Text:='Special Mode 4';
MessageHandler.Msg.Color:=Color.yellow;
MessageHandler.Msg.Station:=1;


MessageHandler(
	Prio:=2, 									(*1=highest, .. , 4=lowest*)
	Btn1Addr:=ADR(MsgOk),			(*Address of Button1 , if Zero then Button is unvisible*)
	Btn2Addr:=ADR(MsgCancel),	(*Address of Button2 , if Zero then Button is unvisible*)
	sVisu:=Visu.Message);


MessageHandler.MessageLine[1].Visible:=TRUE;
MessageHandler.MessageLine[1].Editable:=TRUE;
MessageHandler.MessageLine[1].Text:='Kamera Programm ';
MessageHandler.MessageLine[1].MsgTypeEnum:=MsgDataTypeDint;
END_ACTION

ACTION Msg_Start_exit:
MsgOk:=FALSE;
MsgCancel:=FALSE;

SpecialModeProgNu:=MessageHandler.MessageLine[1].MsgInt;
END_ACTION

ACTION SeqEnd_action:
IF 	State=STATE_RUN THEN
	SFCTime:=TIME_TO_DINT(TIME()-SFCTimeStart);
	State:=STATE_OK;
END_IF

IF 	NOT Start THEN
	State:=STATE_WAIT;
END_IF
END_ACTION
END_PROGRAM

(* POU Stations/ST_00/ST00_SFCs/_SpecialModeSFCs/SpecialMode05, SFC *)
PROGRAM SpecialMode05 (*Used for: xxxx *)
(* Date:     Author:   *)

VAR_OUTPUT
	SFCCurrentPOU		: STRING:='SpecialMode05';
	SFCCurrentStep	: STRING:='';
	SFCTime					:	DINT;
  State   				:	DINT;
  Result  				:	DINT;

	ConveyorOn				: BOOL;

END_VAR
VAR_INPUT
	Start						:	BOOL;
END_VAR
VAR
	MsgOK				:	BOOL;
	MsgCancel		:	BOOL;
	SFCRun					:	BOOL;
	SFCTimeStart		:	TIME;

	(* Userdefinded area *)

END_VAR
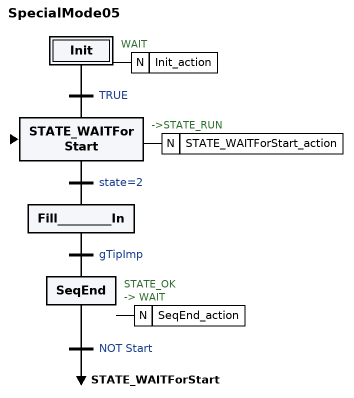
INITIAL_STEP Init: (* WAIT *)
	Init_action(N);
END_STEP
TRANSITION FROM Init TO STATE_WAITForStart := TRUE;
END_TRANSITION
STEP STATE_WAITForStart: (* ->STATE_RUN *)
	STATE_WAITForStart_action(N);
END_STEP
TRANSITION FROM STATE_WAITForStart TO Fill_________In := state=2;
END_TRANSITION
STEP Fill_________In:
END_STEP
TRANSITION FROM Fill_________In TO SeqEnd := gTipImp;
END_TRANSITION
STEP SeqEnd: (* STATE_OK / -> WAIT *)
	SeqEnd_action(N);
END_STEP
TRANSITION FROM SeqEnd TO STATE_WAITForStart := NOT Start;
END_TRANSITION

ACTION Init_action:
Start:=FALSE;
State:=STATE_WAIT;
END_ACTION

ACTION STATE_WAITForStart_action:
IF Start=TRUE
THEN
	State:=STATE_RUN;
	Result:=RESULT_NON;
	SFCTimeStart:=TIME();
(*ELSE*)
END_IF
END_ACTION

ACTION SeqEnd_action:
IF 	State=STATE_RUN THEN
	SFCTime:=TIME_TO_DINT(TIME()-SFCTimeStart);
	State:=STATE_OK;
END_IF

IF 	NOT Start THEN
	State:=STATE_WAIT;
END_IF
END_ACTION
END_PROGRAM

(* POU Stations/ST_00/ST00_SFCs/_SpecialModeSFCs/SpecialMode07, SFC *)
PROGRAM SpecialMode07 (*Used for: xxxx *)
(* Date:     Author:   *)

VAR_OUTPUT
	SFCCurrentPOU		: STRING:='SpecialMode07';
	SFCCurrentStep	: STRING:='';
	SFCTime					:	DINT;
  State   				:	DINT;
  Result  				:	DINT;
END_VAR
VAR_INPUT
	Start						:	BOOL;
END_VAR
VAR
	MsgOK				:	BOOL;
	MsgCancel		:	BOOL;
	SFCRun					:	BOOL;
	SFCTimeStart		:	TIME;
  Delay         :TON;

	(* Userdefinded area *)


END_VAR
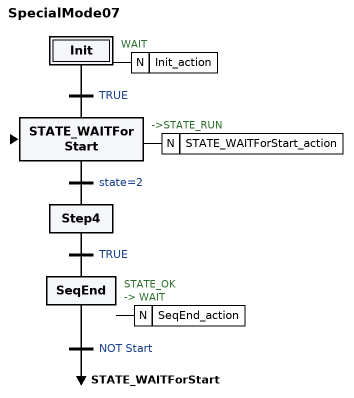
INITIAL_STEP Init: (* WAIT *)
	Init_action(N);
END_STEP
TRANSITION FROM Init TO STATE_WAITForStart := TRUE;
END_TRANSITION
STEP STATE_WAITForStart: (* ->STATE_RUN *)
	STATE_WAITForStart_action(N);
END_STEP
TRANSITION FROM STATE_WAITForStart TO Step4 := state=2;
END_TRANSITION
STEP Step4:
END_STEP
TRANSITION FROM Step4 TO SeqEnd := TRUE;
END_TRANSITION
STEP SeqEnd: (* STATE_OK / -> WAIT *)
	SeqEnd_action(N);
END_STEP
TRANSITION FROM SeqEnd TO STATE_WAITForStart := NOT Start;
END_TRANSITION

ACTION Init_action:
Start:=FALSE;
State:=STATE_WAIT;
END_ACTION

ACTION STATE_WAITForStart_action:
IF Start=TRUE
THEN
	State:=STATE_RUN;
	Result:=RESULT_NON;
	SFCTimeStart:=TIME();
(*ELSE*)
END_IF
END_ACTION

ACTION SeqEnd_action:
IF 	State=STATE_RUN THEN
	SFCTime:=TIME_TO_DINT(TIME()-SFCTimeStart);
	State:=STATE_OK;
END_IF

IF 	NOT Start THEN
	State:=STATE_WAIT;
END_IF
END_ACTION
END_PROGRAM

(* POU Stations/ST_00/ST00_SFCs/_SpecialModeSFCs/SpecialMode08, SFC *)
PROGRAM SpecialMode08 (*Used for: xxxx *)
(* Date:     Author:   *)

VAR_OUTPUT
	SFCCurrentPOU		: STRING:='SpecialMode08';
	SFCCurrentStep	: STRING:='';
	SFCTime					:	DINT;
  State   				:	DINT;
  Result  				:	DINT;
END_VAR
VAR_INPUT
	Start						:	BOOL;
END_VAR
VAR
	MsgOK				:	BOOL;
	MsgCancel		:	BOOL;
	SFCRun					:	BOOL;
	SFCTimeStart		:	TIME;

	(* Userdefinded area *)
	TestDint1:DINT:=12;
	TestDint2:DINT:=34;
	IntPosIdx:	DINT;

END_VAR
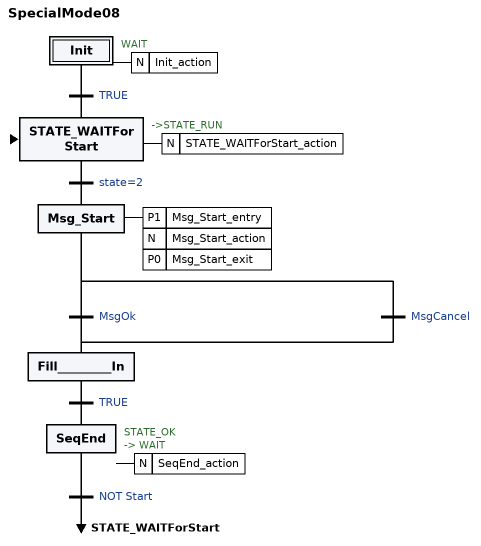
INITIAL_STEP Init: (* WAIT *)
	Init_action(N);
END_STEP
TRANSITION FROM Init TO STATE_WAITForStart := TRUE;
END_TRANSITION
STEP STATE_WAITForStart: (* ->STATE_RUN *)
	STATE_WAITForStart_action(N);
END_STEP
TRANSITION FROM STATE_WAITForStart TO Msg_Start := state=2;
END_TRANSITION
STEP Msg_Start:
	Msg_Start_entry(P1);
	Msg_Start_action(N);
	Msg_Start_exit(P0);
END_STEP
TRANSITION FROM Msg_Start TO Fill_________In := MsgOk;
END_TRANSITION
TRANSITION FROM Msg_Start TO Fill_________In := MsgCancel;
END_TRANSITION
STEP Fill_________In:
END_STEP
TRANSITION FROM Fill_________In TO SeqEnd := TRUE;
END_TRANSITION
STEP SeqEnd: (* STATE_OK / -> WAIT *)
	SeqEnd_action(N);
END_STEP
TRANSITION FROM SeqEnd TO STATE_WAITForStart := NOT Start;
END_TRANSITION

ACTION Init_action:
Start:=FALSE;
State:=STATE_WAIT;
END_ACTION

ACTION STATE_WAITForStart_action:
IF Start=TRUE
THEN
	State:=STATE_RUN;
	Result:=RESULT_NON;
	SFCTimeStart:=TIME();
(*ELSE*)
END_IF
END_ACTION

ACTION Msg_Start_entry:
MessageHandler.ClearMessageLines(sVisu:=Visu.Message);
IntPosIdx:=1;
END_ACTION

ACTION Msg_Start_action:
MessageHandler.Msg.ID:='PM53';
MessageHandler.Msg.Name:='SpecialMode08_Start';
MessageHandler.Msg.Text:='Teilautomatik Ablauf08: Test Messagehandler';
MessageHandler.Msg.Color:=Color.yellow;
MessageHandler.Msg.Station:=1;


MessageHandler(
	Prio:=2, 									(*1=highest, .. , 4=lowest*)
	Btn1Addr:=ADR(MsgOk),			(*Address of Button1 , if Zero then Button is unvisible*)
	Btn2Addr:=ADR(MsgCancel),	(*Address of Button2 , if Zero then Button is unvisible*)
	sVisu:=Visu.Message);


MessageHandler.MessageLine[1].Visible:=TRUE;
MessageHandler.MessageLine[1].Editable:=TRUE;
MessageHandler.MessageLine[1].Text:='TestZeile1';
MessageHandler.MessageLine[1].MsgInt:=TestDint1;
MessageHandler.MessageLine[1].MsgTypeEnum:=MsgDataTypeDint;

MessageHandler.MessageLine[2].Visible:=TRUE;
MessageHandler.MessageLine[2].Editable:=TRUE;
MessageHandler.MessageLine[2].Text:='TestZeile2';
MessageHandler.MessageLine[2].MsgInt:=TestDint2;
MessageHandler.MessageLine[2].MsgTypeEnum:=MsgDataTypeDint;
END_ACTION

ACTION Msg_Start_exit:
MsgOk:=FALSE;
MsgCancel:=FALSE;

TestDint1:=MessageHandler.MessageLine[1].MsgInt;
TestDint2:=MessageHandler.MessageLine[2].MsgInt;
END_ACTION

ACTION SeqEnd_action:
IF 	State=STATE_RUN THEN
	SFCTime:=TIME_TO_DINT(TIME()-SFCTimeStart);
	State:=STATE_OK;
END_IF


IF 	NOT Start THEN
	State:=STATE_WAIT;
END_IF
END_ACTION
END_PROGRAM

(* POU Stations/ST_00/ST00_SFCs/HomePositionSFC, SFC *)
PROGRAM HomePositionSFC


VAR_OUTPUT
	SFCCurrentPOU		: STRING:='HomePositionSFC';
	SFCCurrentStep		: STRING:='';
	SFCTime				: DINT;
	State   			: StateObject	:= STATE_WAIT;
	Result  			: StateResult;
END_VAR
VAR_INPUT
	Start				: BOOL;
END_VAR
VAR
	MsgOK				: BOOL;
	MsgCancel			: BOOL;
	SFCRun				: BOOL;
	SFCTimeStart		: TIME;
	Error				: ErrorStruct;
	(* Userdefinded area *)
	SFCRun01			: BOOL;
	SFCRun02			: BOOL;
	SFCRun03			: BOOL;
	SFCRun04			: BOOL;
	SFCRun05			: BOOL;
	SFCRun08			: BOOL;
	idx					: INT;


END_VAR
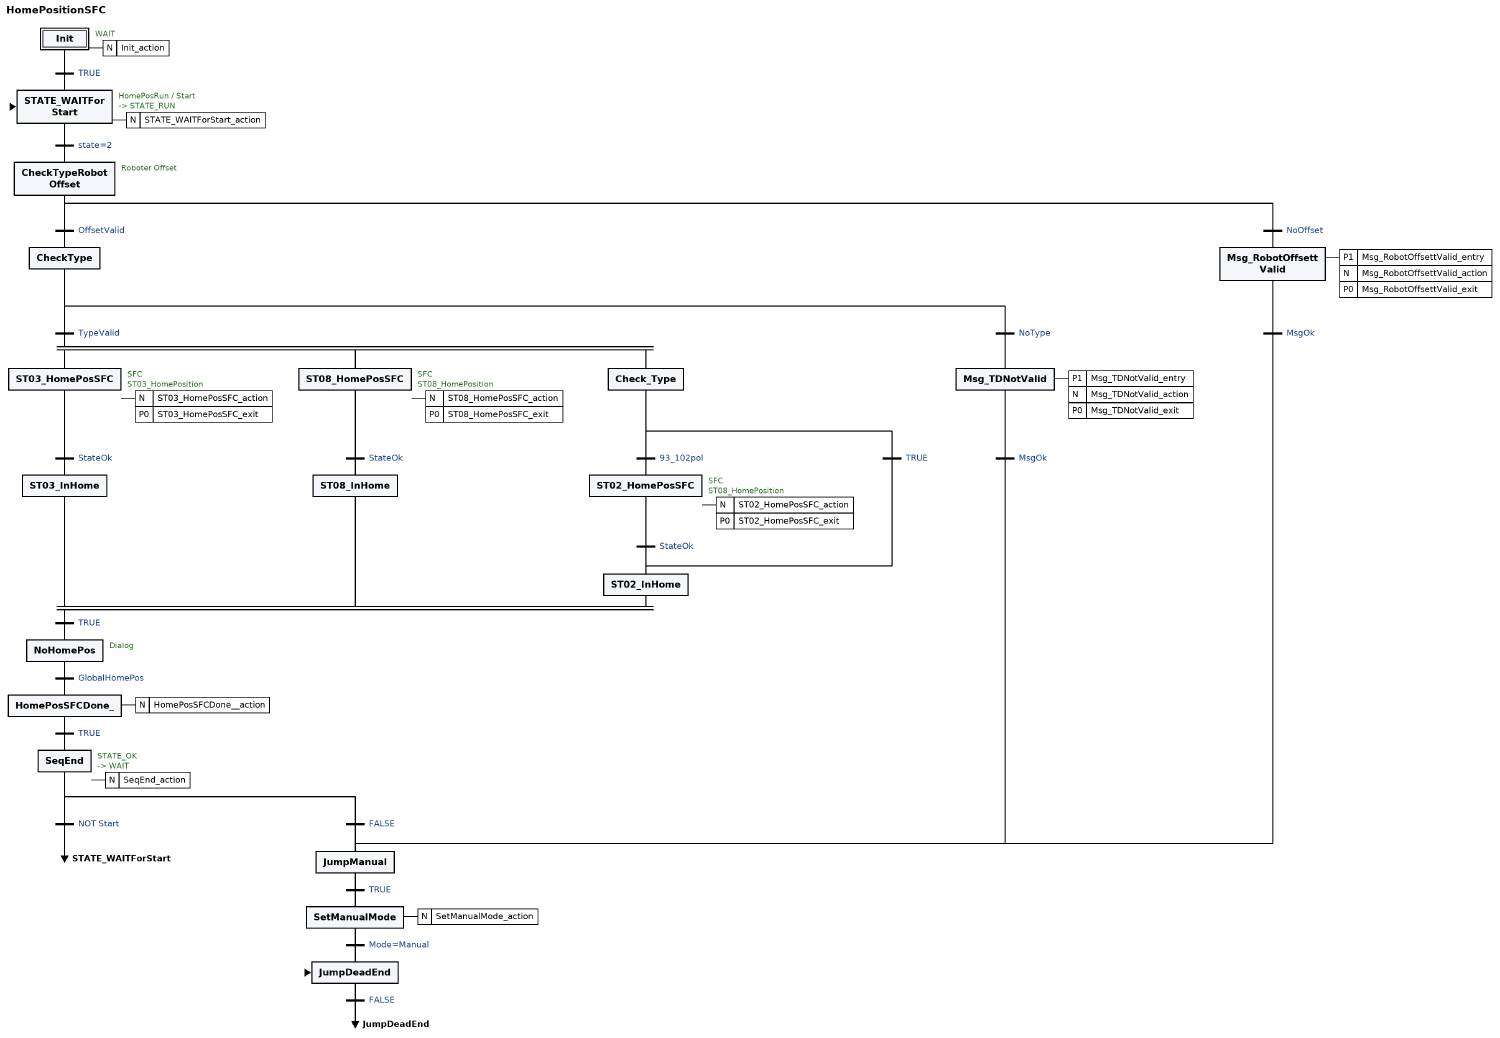
INITIAL_STEP Init: (* WAIT *)
	Init_action(N);
END_STEP
TRANSITION FROM Init TO STATE_WAITForStart := TRUE;
END_TRANSITION
STEP STATE_WAITForStart: (* HomePosRun / Start / -> STATE_RUN *)
	STATE_WAITForStart_action(N);
END_STEP
TRANSITION FROM STATE_WAITForStart TO CheckTypeRobotOffset := state=2;
END_TRANSITION
STEP CheckTypeRobotOffset: (* Roboter Offset *)
END_STEP
TRANSITION FROM CheckTypeRobotOffset TO CheckType := OffsetValid;
END_TRANSITION
TRANSITION FROM CheckTypeRobotOffset TO Msg_RobotOffsettValid := NoOffset;
END_TRANSITION
STEP CheckType:
END_STEP
TRANSITION FROM CheckType TO (ST03_HomePosSFC, ST08_HomePosSFC, Check_Type) := TypeValid;
END_TRANSITION
TRANSITION FROM CheckType TO Msg_TDNotValid := NoType;
END_TRANSITION
STEP Msg_TDNotValid:
	Msg_TDNotValid_entry(P1);
	Msg_TDNotValid_action(N);
	Msg_TDNotValid_exit(P0);
END_STEP
TRANSITION FROM Msg_TDNotValid TO JumpManual := MsgOk;
END_TRANSITION
STEP Msg_RobotOffsettValid:
	Msg_RobotOffsettValid_entry(P1);
	Msg_RobotOffsettValid_action(N);
	Msg_RobotOffsettValid_exit(P0);
END_STEP
TRANSITION FROM Msg_RobotOffsettValid TO JumpManual := MsgOk;
END_TRANSITION
STEP ST03_HomePosSFC: (* SFC / ST03_HomePosition *)
	ST03_HomePosSFC_action(N);
	ST03_HomePosSFC_exit(P0);
END_STEP
TRANSITION FROM ST03_HomePosSFC TO ST03_InHome := StateOk;
END_TRANSITION
STEP ST03_InHome:
END_STEP
STEP ST08_HomePosSFC: (* SFC / ST08_HomePosition *)
	ST08_HomePosSFC_action(N);
	ST08_HomePosSFC_exit(P0);
END_STEP
TRANSITION FROM ST08_HomePosSFC TO ST08_InHome := StateOk;
END_TRANSITION
STEP ST08_InHome:
END_STEP
STEP Check_Type:
END_STEP
TRANSITION FROM Check_Type TO ST02_HomePosSFC := 93_102pol;
END_TRANSITION
TRANSITION FROM Check_Type TO ST02_InHome := TRUE;
END_TRANSITION
STEP ST02_HomePosSFC: (* SFC / ST08_HomePosition *)
	ST02_HomePosSFC_action(N);
	ST02_HomePosSFC_exit(P0);
END_STEP
TRANSITION FROM ST02_HomePosSFC TO ST02_InHome := StateOk;
END_TRANSITION
STEP ST02_InHome:
END_STEP
TRANSITION FROM (ST03_InHome, ST08_InHome, ST02_InHome) TO NoHomePos := TRUE;
END_TRANSITION
STEP NoHomePos: (* Dialog *)
END_STEP
TRANSITION FROM NoHomePos TO HomePosSFCDone_ := GlobalHomePos;
END_TRANSITION
STEP HomePosSFCDone_:
	HomePosSFCDone__action(N);
END_STEP
TRANSITION FROM HomePosSFCDone_ TO SeqEnd := TRUE;
END_TRANSITION
STEP SeqEnd: (* STATE_OK / -> WAIT *)
	SeqEnd_action(N);
END_STEP
TRANSITION FROM SeqEnd TO STATE_WAITForStart := NOT Start;
END_TRANSITION
TRANSITION FROM SeqEnd TO JumpManual := FALSE;
END_TRANSITION
STEP JumpManual:
END_STEP
TRANSITION FROM JumpManual TO SetManualMode := TRUE;
END_TRANSITION
STEP SetManualMode:
	SetManualMode_action(N);
END_STEP
TRANSITION FROM SetManualMode TO JumpDeadEnd := Mode=Manual;
END_TRANSITION
STEP JumpDeadEnd:
END_STEP
TRANSITION FROM JumpDeadEnd TO JumpDeadEnd := FALSE;
END_TRANSITION

ACTION Init_action:
Start:=FALSE;
State:=STATE_WAIT;
END_ACTION

ACTION STATE_WAITForStart_action:
IF	(ModeSelect.Mode=MODE_HOME_POS_RUN OR
	Start) AND
	NOT PLC_PRG.GlobalHomePos THEN
	State:=STATE_RUN;
	Result:=RESULT_NON;
	SFCTimeStart:=TIME();
END_IF

SFCRun		:=FALSE;
SFCRun01	:=FALSE;
SFCRun02	:=FALSE;
SFCRun03	:=FALSE;
SFCRun04	:=FALSE;
SFCRun05	:=FALSE;
END_ACTION

ACTION Msg_TDNotValid_entry:
FOR idx:=1 TO 8
DO
	MessageHandler.MessageLine[idx].Visible:=FALSE;
	MessageHandler.MessageLine[idx].Editable:=FALSE;
	MessageHandler.MessageLine[idx].Text:='';
	MessageHandler.MessageLine[idx].MsgInt:=0;
	MessageHandler.MessageLine[idx].MsgTypeEnum:=MsgDataTypeDint;

END_FOR
END_ACTION

ACTION Msg_TDNotValid_action:
MessageHandler.Msg.ID:='PM10';
MessageHandler.Msg.Name:='TDNotValid';
MessageHandler.Msg.Text:='Typdaten nicht gültig, bitte laden!';
MessageHandler.Msg.Text:= CONCAT(MessageHandler.Msg.Text,'$r --> weiter mit <OK>');
MessageHandler.Msg.Color:=Color.yellow;
MessageHandler.Msg.Station:=0;
MessageHandler.MsgButton1Text:='continue';

MessageHandler(
	Prio:=1, 						(*1=highest, .. , 4=lowest*)
	Btn1Addr:=ADR(MsgOk),		(*Address of Button1 , if Zero then Button is unvisible*)
	Btn2Addr:=0,					(*Address of Button2 , if Zero then Button is unvisible*)
	sVisu:=Visu.Message);
END_ACTION

ACTION Msg_TDNotValid_exit:
MsgOk:=FALSE;
MsgCancel:=FALSE;
END_ACTION

ACTION Msg_RobotOffsettValid_entry:
MessageHandler.ClearMessageLines(sVisu:=Visu.Message);
END_ACTION

ACTION Msg_RobotOffsettValid_action:
MessageHandler.Msg.ID:='PM11';
MessageHandler.Msg.Name:='TDRoffsetbotOValid';
MessageHandler.Msg.Text:='Typdaten Roboter Offset nicht gültig, bitte laden!';
MessageHandler.Msg.Text:= CONCAT(MessageHandler.Msg.Text,'$r --> weiter mit <OK>');

MessageHandler.Msg.Color:=Color.yellow;
MessageHandler.Msg.Station:=0;


MessageHandler(
	Prio:=1, 								(*1=highest, .. , 4=lowest*)
	Btn1Addr:=ADR(MsgOk),		(*Address of Button1 , if Zero then Button is unvisible*)
	Btn2Addr:=0,						(*Address of Button2 , if Zero then Button is unvisible*)
	sVisu:=Visu.Message);
END_ACTION

ACTION Msg_RobotOffsettValid_exit:
MsgOk:=FALSE;
MsgCancel:=FALSE;
END_ACTION

ACTION ST03_HomePosSFC_action:
IF ST03_HomePosition.State=STATE_WAIT
THEN
	ST03_HomePosition(Start:=TRUE);

	SFCRun03:=TRUE;
(*ELSE*)
END_IF
END_ACTION

ACTION ST03_HomePosSFC_exit:
ST03_HomePosition.Start:=FALSE;
SFCRun03:=FALSE;
END_ACTION

ACTION ST08_HomePosSFC_action:
IF ST08_HomePosition.State=STATE_WAIT
THEN
	SFCRun08:=TRUE;
	ST08_HomePosition.Start:=TRUE;


(*ELSE*)
END_IF
END_ACTION

ACTION ST08_HomePosSFC_exit:
ST08_HomePosition.Start:=FALSE;
SFCRun08:=FALSE;
END_ACTION

ACTION ST02_HomePosSFC_action:
IF ST02_HomePosition.State=STATE_WAIT THEN
	ST02_HomePosition.Start:=TRUE;
	SFCRun02:=TRUE;
END_IF
END_ACTION

ACTION ST02_HomePosSFC_exit:
ST02_HomePosition.Start:=FALSE;
SFCRun02:=FALSE;
END_ACTION

ACTION HomePosSFCDone__action:
gHomePosSFCDone:=TRUE;
END_ACTION

ACTION SeqEnd_action:
IF 	NOT Start THEN
	State:=STATE_WAIT;
END_IF
END_ACTION

ACTION SetManualMode_action:
ModeSelect.AskForManual:=TRUE;
END_ACTION

TRANSITION OffsetValid:
   gRobotOffset > 0
(*OR gRobotOffset =1000
OR gRobotOffset =2000
OR gRobotOffset =3000
OR gRobotOffset =4000
OR gRobotOffset =5000
OR gRobotOffset =6000
OR gRobotOffset =7000
OR gRobotOffset =19000
OR gRobotOffset =25000
OR gRobotOffset =26000
OR gRobotOffset =27000
OR gRobotOffset =28000
OR gRobotOffset =29000
OR gRobotOffset =30000
OR gRobotOffset =35000*)
END_TRANSITION

TRANSITION TypeValid:
gTypeDataValid
END_TRANSITION

TRANSITION NoType:
TRUE
END_TRANSITION

TRANSITION NoOffset:
TRUE
END_TRANSITION

TRANSITION StateOk:
		SFCRun03=TRUE
AND ST03_HomePosition.State=STATE_OK
END_TRANSITION

TRANSITION StateOk:
		SFCRun08=TRUE
AND ST08_HomePosition.State=STATE_OK
END_TRANSITION

TRANSITION 93_102pol:
gTypeCode=4991 OR 	(*102pol*)
gTypeCode=312		(*93pol*)
END_TRANSITION

TRANSITION StateOk:
SFCRun02 AND
ST02_HomePosition.State=STATE_OK
END_TRANSITION

TRANSITION GlobalHomePos:
PLC_PRG.GlobalHomePos
END_TRANSITION

TRANSITION Mode=Manual:
ModeSelect.Mode=MODE_MANUAL
END_TRANSITION
END_PROGRAM

(* POU Stations/ST_03_Ruestsaetze/ST_03_SFCs/ST03_HomePosition, SFC *)
PROGRAM ST03_HomePosition

VAR_OUTPUT
	SFCCurrentPOU		: STRING:='ST03_HomePosition';
	SFCCurrentStep		: STRING:='';
	SFCTime				: DINT;
	State   			: StateObject	:= STATE_WAIT;
	Result  			: StateResult;

END_VAR
VAR_INPUT
	Start				: BOOL;
END_VAR
VAR
	MsgOK				: BOOL;
	MsgCancel			: BOOL;
	SFCRun				: BOOL;
	SFCTimeStart		: TIME;
	(* Userdefinded area *)

END_VAR
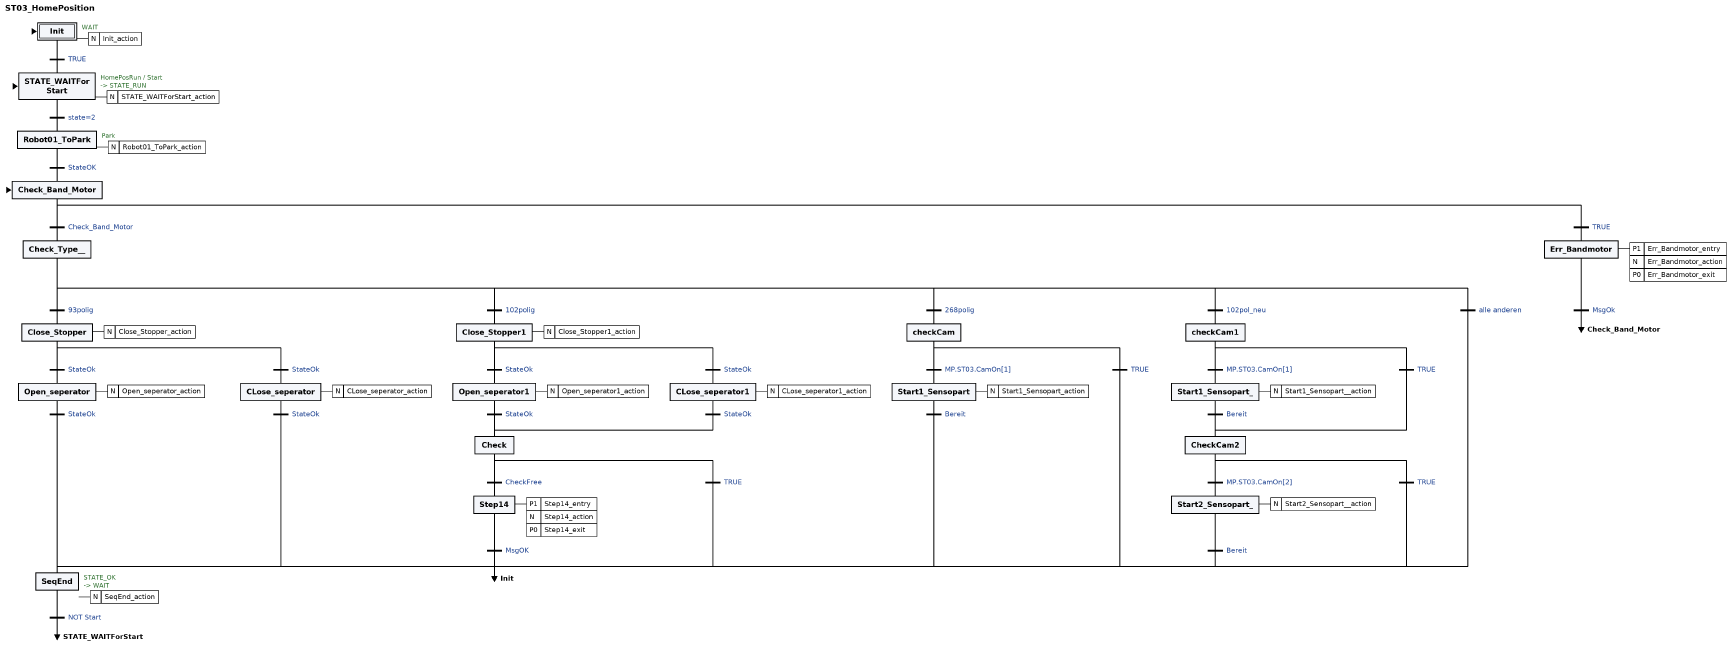
INITIAL_STEP Init: (* WAIT *)
	Init_action(N);
END_STEP
TRANSITION FROM Init TO STATE_WAITForStart := TRUE;
END_TRANSITION
STEP STATE_WAITForStart: (* HomePosRun / Start / -> STATE_RUN *)
	STATE_WAITForStart_action(N);
END_STEP
TRANSITION FROM STATE_WAITForStart TO Robot01_ToPark := state=2;
END_TRANSITION
STEP Robot01_ToPark: (* Park *)
	Robot01_ToPark_action(N);
END_STEP
TRANSITION FROM Robot01_ToPark TO Check_Band_Motor := StateOK;
END_TRANSITION
STEP Check_Band_Motor:
END_STEP
TRANSITION FROM Check_Band_Motor TO Check_Type__ := Check_Band_Motor;
END_TRANSITION
TRANSITION FROM Check_Band_Motor TO Err_Bandmotor := TRUE;
END_TRANSITION
STEP Err_Bandmotor:
	Err_Bandmotor_entry(P1);
	Err_Bandmotor_action(N);
	Err_Bandmotor_exit(P0);
END_STEP
TRANSITION FROM Err_Bandmotor TO Check_Band_Motor := MsgOk;
END_TRANSITION
STEP Check_Type__:
END_STEP
TRANSITION FROM Check_Type__ TO Close_Stopper := 93polig;
END_TRANSITION
TRANSITION FROM Check_Type__ TO Close_Stopper1 := 102polig;
END_TRANSITION
TRANSITION FROM Check_Type__ TO checkCam := 268polig;
END_TRANSITION
TRANSITION FROM Check_Type__ TO checkCam1 := 102pol_neu;
END_TRANSITION
TRANSITION FROM Check_Type__ TO SeqEnd := alle anderen;
END_TRANSITION
STEP Close_Stopper:
	Close_Stopper_action(N);
END_STEP
TRANSITION FROM Close_Stopper TO Open_seperator := StateOk;
END_TRANSITION
TRANSITION FROM Close_Stopper TO CLose_seperator := StateOk;
END_TRANSITION
STEP Open_seperator:
	Open_seperator_action(N);
END_STEP
TRANSITION FROM Open_seperator TO SeqEnd := StateOk;
END_TRANSITION
STEP CLose_seperator:
	CLose_seperator_action(N);
END_STEP
TRANSITION FROM CLose_seperator TO SeqEnd := StateOk;
END_TRANSITION
STEP Close_Stopper1:
	Close_Stopper1_action(N);
END_STEP
TRANSITION FROM Close_Stopper1 TO Open_seperator1 := StateOk;
END_TRANSITION
TRANSITION FROM Close_Stopper1 TO CLose_seperator1 := StateOk;
END_TRANSITION
STEP Open_seperator1:
	Open_seperator1_action(N);
END_STEP
TRANSITION FROM Open_seperator1 TO Check := StateOk;
END_TRANSITION
STEP CLose_seperator1:
	CLose_seperator1_action(N);
END_STEP
TRANSITION FROM CLose_seperator1 TO Check := StateOk;
END_TRANSITION
STEP Check:
END_STEP
TRANSITION FROM Check TO Step14 := CheckFree;
END_TRANSITION
TRANSITION FROM Check TO SeqEnd := TRUE;
END_TRANSITION
STEP Step14:
	Step14_entry(P1);
	Step14_action(N);
	Step14_exit(P0);
END_STEP
TRANSITION FROM Step14 TO Init := MsgOK;
END_TRANSITION
STEP checkCam:
END_STEP
TRANSITION FROM checkCam TO Start1_Sensopart := MP.ST03.CamOn[1];
END_TRANSITION
TRANSITION FROM checkCam TO SeqEnd := TRUE;
END_TRANSITION
STEP Start1_Sensopart:
	Start1_Sensopart_action(N);
END_STEP
TRANSITION FROM Start1_Sensopart TO SeqEnd := Bereit;
END_TRANSITION
STEP checkCam1:
END_STEP
TRANSITION FROM checkCam1 TO Start1_Sensopart_ := MP.ST03.CamOn[1];
END_TRANSITION
TRANSITION FROM checkCam1 TO CheckCam2 := TRUE;
END_TRANSITION
STEP Start1_Sensopart_:
	Start1_Sensopart__action(N);
END_STEP
TRANSITION FROM Start1_Sensopart_ TO CheckCam2 := Bereit;
END_TRANSITION
STEP CheckCam2:
END_STEP
TRANSITION FROM CheckCam2 TO Start2_Sensopart_ := MP.ST03.CamOn[2];
END_TRANSITION
TRANSITION FROM CheckCam2 TO SeqEnd := TRUE;
END_TRANSITION
STEP Start2_Sensopart_:
	Start2_Sensopart__action(N);
END_STEP
TRANSITION FROM Start2_Sensopart_ TO SeqEnd := Bereit;
END_TRANSITION
STEP SeqEnd: (* STATE_OK / -> WAIT *)
	SeqEnd_action(N);
END_STEP
TRANSITION FROM SeqEnd TO STATE_WAITForStart := NOT Start;
END_TRANSITION

ACTION Init_action:
Start:=FALSE;
State:=STATE_WAIT;
END_ACTION

ACTION STATE_WAITForStart_action:
IF	( Start = TRUE )
THEN
	State:=STATE_RUN;
	Result:=RESULT_NON;
	SFCTimeStart:=TIME();
ELSE
	;
END_IF
END_ACTION

ACTION Robot01_ToPark_action:
Robot01.PosNo:=POS_PARK;
Robot01.PosOffset:=gRobotOffset;
Robot01.Override:=MP.ST00.Override;
Robot01.SetToolOn:=FALSE;
Robot01.SetToolOff:=FALSE;
Robot01.ExecuteMove:=TRUE;
END_ACTION

ACTION Err_Bandmotor_entry:
MessageHandler.ClearMessageLines(sVisu:=Visu.Message);
END_ACTION

ACTION Err_Bandmotor_action:
MessageHandler.Msg.ID:='PM100';
MessageHandler.Msg.Name:='Fehler Bandmotor';
MessageHandler.Msg.Text:='Fehler Bandmotor';
MessageHandler.Msg.Color:=Color.red;
MessageHandler.Msg.Station:=1;


MessageHandler(
	Prio:=2, 							(*1=highest, .. , 4=lowest*)
	Btn1Addr:=ADR(MsgOk),			(*Address of Button1 , if Zero then Button is unvisible*)
	Btn2Addr:=,						(*Address of Button2 , if Zero then Button is unvisible*)
	sVisu:=Visu.Message);
END_ACTION

ACTION Err_Bandmotor_exit:
MsgOk:=FALSE;
MsgCancel:=FALSE;
ST03_51_M1.Reset:=TRUE;
END_ACTION

ACTION Close_Stopper_action:
ST00_74_Y2_4.MoveInit:=TRUE;
END_ACTION

ACTION Open_seperator_action:
ST00_74_Y2_5.MoveInit:=TRUE;
END_ACTION

ACTION CLose_seperator_action:
ST00_74_Y2_5.MoveWork:=TRUE;
END_ACTION

ACTION Close_Stopper1_action:
ST00_74_Y2_4.MoveInit:=TRUE;
END_ACTION

ACTION Open_seperator1_action:
ST00_74_Y2_5.MoveInit:=TRUE;
END_ACTION

ACTION CLose_seperator1_action:
ST00_74_Y2_5.MoveWork:=TRUE;
END_ACTION

ACTION Step14_entry:
MessageHandler.ClearMessageLines(sVisu:=Visu.Message);
END_ACTION

ACTION Step14_action:
MessageHandler.Msg.ID:='PM102';
MessageHandler.Msg.Name:='Vereinzler beide Positionen besetzt';
MessageHandler.Msg.Text:='Vereinzler beide Positionen besetzt';
MessageHandler.Msg.Color:=Color.red;
MessageHandler.Msg.Station:=1;


MessageHandler(
	Prio:=2, 							(*1=highest, .. , 4=lowest*)
	Btn1Addr:=ADR(MsgOk),			(*Address of Button1 , if Zero then Button is unvisible*)
	Btn2Addr:=,						(*Address of Button2 , if Zero then Button is unvisible*)
	sVisu:=Visu.Message);
END_ACTION

ACTION Step14_exit:
MsgOk:=FALSE;
MsgCancel:=FALSE;
END_ACTION

ACTION Start1_Sensopart_action:
ST03_8_100_A1.JobNo := TD.Sensopart_CamProgNo ;
ST03_8_100_A1.st_ctrl_in.b_init := TRUE;
END_ACTION

ACTION Start1_Sensopart__action:
ST03_8_100_A1.JobNo := TD.Sensopart_CamProgNo ;
ST03_8_100_A1.st_ctrl_in.b_init := TRUE;
END_ACTION

ACTION Start2_Sensopart__action:
ST03_8_103_A1.JobNo := TD.Sensopart2_CamProgNo ;
ST03_8_103_A1.st_ctrl_in.b_init := TRUE;
END_ACTION

ACTION SeqEnd_action:
IF 	State=STATE_RUN THEN
	SFCTime:=TIME_TO_DINT(TIME()-SFCTimeStart);
	State:=STATE_OK;
END_IF

IF 	NOT Start THEN
	State:=STATE_WAIT;
END_IF
END_ACTION

TRANSITION StateOK:
Robot01.State=STATE_OK
END_TRANSITION

TRANSITION Check_Band_Motor:
NOT ST03_51_M1.Error_ (*AND
ST03_51_M1.On*)
END_TRANSITION

TRANSITION 93polig:
gTypeCode=312	(*93pol*)
END_TRANSITION

TRANSITION StateOk:
ST00_74_Y2_4.State=STATE_OK AND
NOT ST00_72_X1_3.BitInToCheck
END_TRANSITION

TRANSITION StateOk:
ST00_74_Y2_5.State=STATE_OK
END_TRANSITION

TRANSITION StateOk:
ST00_74_Y2_4.State=STATE_OK
END_TRANSITION

TRANSITION StateOk:
ST00_74_Y2_5.State=STATE_OK
END_TRANSITION

TRANSITION 102polig:
gTypeCode=4991	(*102pol*)
END_TRANSITION

TRANSITION StateOk:
ST00_74_Y2_4.State=STATE_OK AND
NOT ST02_FDB_80_B02.BitInToCheck
END_TRANSITION

TRANSITION StateOk:
ST00_74_Y2_5.State=STATE_OK
END_TRANSITION

TRANSITION StateOk:
ST00_74_Y2_4.State=STATE_OK
END_TRANSITION

TRANSITION StateOk:
ST00_74_Y2_5.State=STATE_OK
END_TRANSITION

TRANSITION CheckFree:
ST02_FDB_80_B02.BitInToCheck AND
ST00_72_X1_3.BitInToCheck
END_TRANSITION

TRANSITION 268polig:
gTypeCode=5841 	(*268pol*)
END_TRANSITION

TRANSITION Bereit:
ST03_8_100_A1.st_ctrl_out.b_bereit (*Kamera Farberkennung Ehternet*)
END_TRANSITION

TRANSITION 102pol_neu:
gTypeCode=4993	(*102pol neu*)
END_TRANSITION

TRANSITION Bereit:
ST03_8_100_A1.st_ctrl_out.b_bereit  (*Kamera Farberkennung Ehternet*)
END_TRANSITION

TRANSITION Bereit:
ST03_8_103_A1.st_ctrl_out.b_bereit  (*Kamera Farberkennung Ehternet*)
END_TRANSITION

TRANSITION alle anderen:
TRUE
END_TRANSITION
END_PROGRAM

(* POU Stations/ST_08_Palettierer/ST_08_SFCs/ST08_HomePosition, SFC *)
PROGRAM ST08_HomePosition


VAR_OUTPUT
	SFCCurrentPOU		: STRING:='ST08_HomePosition';
	SFCCurrentStep		: STRING:='';
	SFCTime				: DINT;
	State   			: StateObject	:= STATE_WAIT;
	Result  			: StateResult;
END_VAR
VAR_INPUT
	Start				: BOOL;
END_VAR
VAR
	MsgOK				: BOOL;
	MsgCancel			: BOOL;
	SFCRun				: BOOL;
	SFCTimeStart		: TIME;
	(* Userdefinded area *)
	MsgString      		:STRING;
	MsgID		      	:STRING(20);
END_VAR
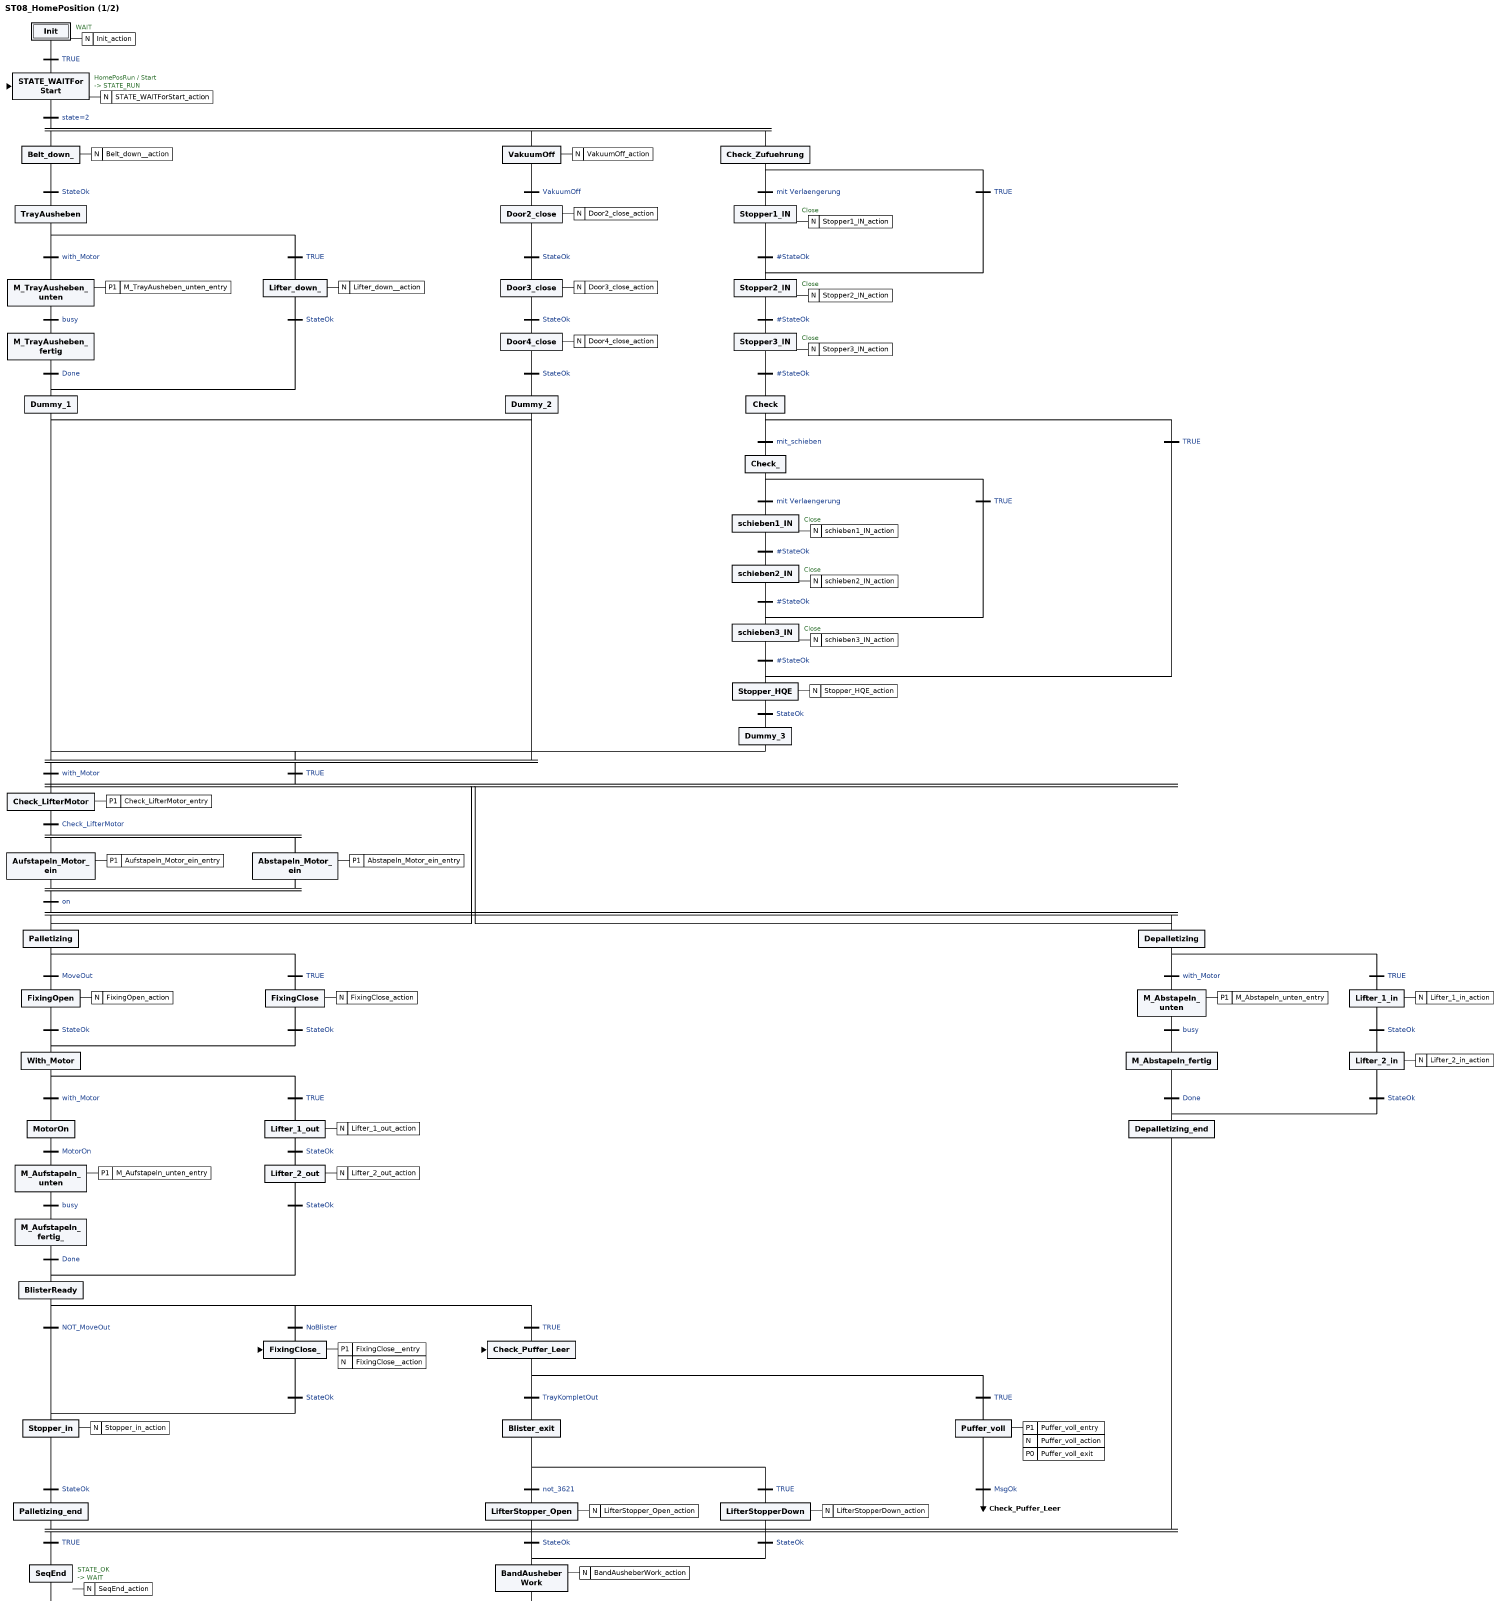
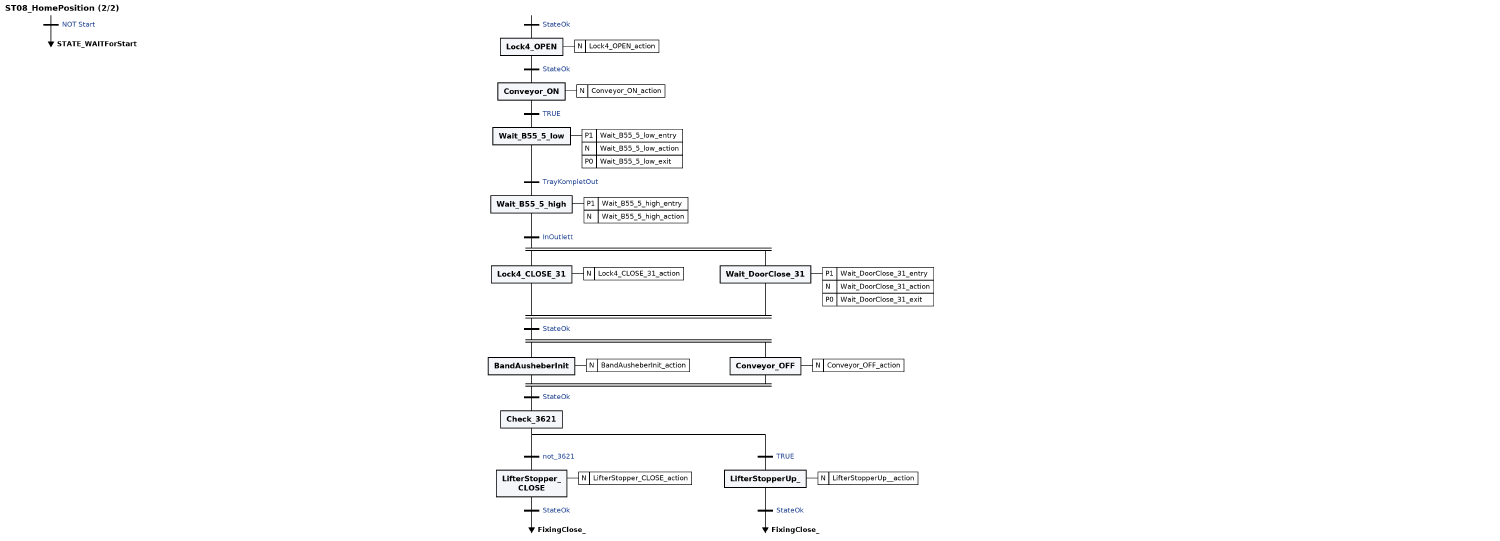
INITIAL_STEP Init: (* WAIT *)
	Init_action(N);
END_STEP
TRANSITION FROM Init TO STATE_WAITForStart := TRUE;
END_TRANSITION
STEP STATE_WAITForStart: (* HomePosRun / Start / -> STATE_RUN *)
	STATE_WAITForStart_action(N);
END_STEP
TRANSITION FROM STATE_WAITForStart TO (Belt_down_, VakuumOff, Check_Zufuehrung) := state=2;
END_TRANSITION
STEP Belt_down_:
	Belt_down__action(N);
END_STEP
TRANSITION FROM Belt_down_ TO TrayAusheben := StateOk;
END_TRANSITION
STEP TrayAusheben:
END_STEP
TRANSITION FROM TrayAusheben TO M_TrayAusheben_unten := with_Motor;
END_TRANSITION
TRANSITION FROM TrayAusheben TO Lifter_down_ := TRUE;
END_TRANSITION
STEP M_TrayAusheben_unten:
	M_TrayAusheben_unten_entry(P1);
END_STEP
TRANSITION FROM M_TrayAusheben_unten TO M_TrayAusheben_fertig := busy;
END_TRANSITION
STEP M_TrayAusheben_fertig:
END_STEP
TRANSITION FROM M_TrayAusheben_fertig TO Dummy_1 := Done;
END_TRANSITION
STEP Lifter_down_:
	Lifter_down__action(N);
END_STEP
TRANSITION FROM Lifter_down_ TO Dummy_1 := StateOk;
END_TRANSITION
STEP Dummy_1:
END_STEP
STEP VakuumOff:
	VakuumOff_action(N);
END_STEP
TRANSITION FROM VakuumOff TO Door2_close := VakuumOff;
END_TRANSITION
STEP Door2_close:
	Door2_close_action(N);
END_STEP
TRANSITION FROM Door2_close TO Door3_close := StateOk;
END_TRANSITION
STEP Door3_close:
	Door3_close_action(N);
END_STEP
TRANSITION FROM Door3_close TO Door4_close := StateOk;
END_TRANSITION
STEP Door4_close:
	Door4_close_action(N);
END_STEP
TRANSITION FROM Door4_close TO Dummy_2 := StateOk;
END_TRANSITION
STEP Dummy_2:
END_STEP
STEP Check_Zufuehrung:
END_STEP
TRANSITION FROM Check_Zufuehrung TO Stopper1_IN := mit Verlaengerung;
END_TRANSITION
TRANSITION FROM Check_Zufuehrung TO Stopper2_IN := TRUE;
END_TRANSITION
STEP Stopper1_IN: (* Close *)
	Stopper1_IN_action(N);
END_STEP
TRANSITION FROM Stopper1_IN TO Stopper2_IN := #StateOk;
END_TRANSITION
STEP Stopper2_IN: (* Close *)
	Stopper2_IN_action(N);
END_STEP
TRANSITION FROM Stopper2_IN TO Stopper3_IN := #StateOk;
END_TRANSITION
STEP Stopper3_IN: (* Close *)
	Stopper3_IN_action(N);
END_STEP
TRANSITION FROM Stopper3_IN TO Check := #StateOk;
END_TRANSITION
STEP Check:
END_STEP
TRANSITION FROM Check TO Check_ := mit_schieben;
END_TRANSITION
TRANSITION FROM Check TO Stopper_HQE := TRUE;
END_TRANSITION
STEP Check_:
END_STEP
TRANSITION FROM Check_ TO schieben1_IN := mit Verlaengerung;
END_TRANSITION
TRANSITION FROM Check_ TO schieben3_IN := TRUE;
END_TRANSITION
STEP schieben1_IN: (* Close *)
	schieben1_IN_action(N);
END_STEP
TRANSITION FROM schieben1_IN TO schieben2_IN := #StateOk;
END_TRANSITION
STEP schieben2_IN: (* Close *)
	schieben2_IN_action(N);
END_STEP
TRANSITION FROM schieben2_IN TO schieben3_IN := #StateOk;
END_TRANSITION
STEP schieben3_IN: (* Close *)
	schieben3_IN_action(N);
END_STEP
TRANSITION FROM schieben3_IN TO Stopper_HQE := #StateOk;
END_TRANSITION
STEP Stopper_HQE:
	Stopper_HQE_action(N);
END_STEP
TRANSITION FROM Stopper_HQE TO Dummy_3 := StateOk;
END_TRANSITION
STEP Dummy_3:
END_STEP
TRANSITION FROM (Dummy_1, Dummy_2, Dummy_3) TO Check_LifterMotor := with_Motor;
END_TRANSITION
TRANSITION FROM (Dummy_1, Dummy_2, Dummy_3) TO (Palletizing, Depalletizing) := TRUE;
END_TRANSITION
STEP Check_LifterMotor:
	Check_LifterMotor_entry(P1);
END_STEP
TRANSITION FROM Check_LifterMotor TO (Aufstapeln_Motor_ein, Abstapeln_Motor_ein) := Check_LifterMotor;
END_TRANSITION
STEP Aufstapeln_Motor_ein:
	Aufstapeln_Motor_ein_entry(P1);
END_STEP
STEP Abstapeln_Motor_ein:
	Abstapeln_Motor_ein_entry(P1);
END_STEP
TRANSITION FROM (Aufstapeln_Motor_ein, Abstapeln_Motor_ein) TO (Palletizing, Depalletizing) := on;
END_TRANSITION
STEP Palletizing:
END_STEP
TRANSITION FROM Palletizing TO FixingOpen := MoveOut;
END_TRANSITION
TRANSITION FROM Palletizing TO FixingClose := TRUE;
END_TRANSITION
STEP FixingOpen:
	FixingOpen_action(N);
END_STEP
TRANSITION FROM FixingOpen TO With_Motor := StateOk;
END_TRANSITION
STEP FixingClose:
	FixingClose_action(N);
END_STEP
TRANSITION FROM FixingClose TO With_Motor := StateOk;
END_TRANSITION
STEP With_Motor:
END_STEP
TRANSITION FROM With_Motor TO MotorOn := with_Motor;
END_TRANSITION
TRANSITION FROM With_Motor TO Lifter_1_out := TRUE;
END_TRANSITION
STEP MotorOn:
END_STEP
TRANSITION FROM MotorOn TO M_Aufstapeln_unten := MotorOn;
END_TRANSITION
STEP M_Aufstapeln_unten:
	M_Aufstapeln_unten_entry(P1);
END_STEP
TRANSITION FROM M_Aufstapeln_unten TO M_Aufstapeln_fertig_ := busy;
END_TRANSITION
STEP M_Aufstapeln_fertig_:
END_STEP
TRANSITION FROM M_Aufstapeln_fertig_ TO BlisterReady := Done;
END_TRANSITION
STEP Lifter_1_out:
	Lifter_1_out_action(N);
END_STEP
TRANSITION FROM Lifter_1_out TO Lifter_2_out := StateOk;
END_TRANSITION
STEP Lifter_2_out:
	Lifter_2_out_action(N);
END_STEP
TRANSITION FROM Lifter_2_out TO BlisterReady := StateOk;
END_TRANSITION
STEP BlisterReady:
END_STEP
TRANSITION FROM BlisterReady TO Stopper_in := NOT_MoveOut;
END_TRANSITION
TRANSITION FROM BlisterReady TO FixingClose_ := NoBlister;
END_TRANSITION
TRANSITION FROM BlisterReady TO Check_Puffer_Leer := TRUE;
END_TRANSITION
STEP FixingClose_:
	FixingClose__entry(P1);
	FixingClose__action(N);
END_STEP
TRANSITION FROM FixingClose_ TO Stopper_in := StateOk;
END_TRANSITION
STEP Check_Puffer_Leer:
END_STEP
TRANSITION FROM Check_Puffer_Leer TO Blister_exit := TrayKompletOut;
END_TRANSITION
TRANSITION FROM Check_Puffer_Leer TO Puffer_voll := TRUE;
END_TRANSITION
STEP Puffer_voll:
	Puffer_voll_entry(P1);
	Puffer_voll_action(N);
	Puffer_voll_exit(P0);
END_STEP
TRANSITION FROM Puffer_voll TO Check_Puffer_Leer := MsgOk;
END_TRANSITION
STEP Blister_exit:
END_STEP
TRANSITION FROM Blister_exit TO LifterStopper_Open := not_3621;
END_TRANSITION
TRANSITION FROM Blister_exit TO LifterStopperDown := TRUE;
END_TRANSITION
STEP LifterStopper_Open:
	LifterStopper_Open_action(N);
END_STEP
TRANSITION FROM LifterStopper_Open TO BandAusheberWork := StateOk;
END_TRANSITION
STEP LifterStopperDown:
	LifterStopperDown_action(N);
END_STEP
TRANSITION FROM LifterStopperDown TO BandAusheberWork := StateOk;
END_TRANSITION
STEP BandAusheberWork:
	BandAusheberWork_action(N);
END_STEP
TRANSITION FROM BandAusheberWork TO Lock4_OPEN := StateOk;
END_TRANSITION
STEP Lock4_OPEN:
	Lock4_OPEN_action(N);
END_STEP
TRANSITION FROM Lock4_OPEN TO Conveyor_ON := StateOk;
END_TRANSITION
STEP Conveyor_ON:
	Conveyor_ON_action(N);
END_STEP
TRANSITION FROM Conveyor_ON TO Wait_B55_5_low := TRUE;
END_TRANSITION
STEP Wait_B55_5_low:
	Wait_B55_5_low_entry(P1);
	Wait_B55_5_low_action(N);
	Wait_B55_5_low_exit(P0);
END_STEP
TRANSITION FROM Wait_B55_5_low TO Wait_B55_5_high := TrayKompletOut;
END_TRANSITION
STEP Wait_B55_5_high:
	Wait_B55_5_high_entry(P1);
	Wait_B55_5_high_action(N);
END_STEP
TRANSITION FROM Wait_B55_5_high TO (Lock4_CLOSE_31, Wait_DoorClose_31) := InOutlett;
END_TRANSITION
STEP Lock4_CLOSE_31:
	Lock4_CLOSE_31_action(N);
END_STEP
STEP Wait_DoorClose_31:
	Wait_DoorClose_31_entry(P1);
	Wait_DoorClose_31_action(N);
	Wait_DoorClose_31_exit(P0);
END_STEP
TRANSITION FROM (Lock4_CLOSE_31, Wait_DoorClose_31) TO (BandAusheberInit, Conveyor_OFF) := StateOk;
END_TRANSITION
STEP BandAusheberInit:
	BandAusheberInit_action(N);
END_STEP
STEP Conveyor_OFF:
	Conveyor_OFF_action(N);
END_STEP
TRANSITION FROM (BandAusheberInit, Conveyor_OFF) TO Check_3621 := StateOk;
END_TRANSITION
STEP Check_3621:
END_STEP
TRANSITION FROM Check_3621 TO LifterStopper_CLOSE := not_3621;
END_TRANSITION
TRANSITION FROM Check_3621 TO LifterStopperUp_ := TRUE;
END_TRANSITION
STEP LifterStopper_CLOSE:
	LifterStopper_CLOSE_action(N);
END_STEP
TRANSITION FROM LifterStopper_CLOSE TO FixingClose_ := StateOk;
END_TRANSITION
STEP LifterStopperUp_:
	LifterStopperUp__action(N);
END_STEP
TRANSITION FROM LifterStopperUp_ TO FixingClose_ := StateOk;
END_TRANSITION
STEP Stopper_in:
	Stopper_in_action(N);
END_STEP
TRANSITION FROM Stopper_in TO Palletizing_end := StateOk;
END_TRANSITION
STEP Palletizing_end:
END_STEP
STEP Depalletizing:
END_STEP
TRANSITION FROM Depalletizing TO M_Abstapeln_unten := with_Motor;
END_TRANSITION
TRANSITION FROM Depalletizing TO Lifter_1_in := TRUE;
END_TRANSITION
STEP M_Abstapeln_unten:
	M_Abstapeln_unten_entry(P1);
END_STEP
TRANSITION FROM M_Abstapeln_unten TO M_Abstapeln_fertig := busy;
END_TRANSITION
STEP M_Abstapeln_fertig:
END_STEP
TRANSITION FROM M_Abstapeln_fertig TO Depalletizing_end := Done;
END_TRANSITION
STEP Lifter_1_in:
	Lifter_1_in_action(N);
END_STEP
TRANSITION FROM Lifter_1_in TO Lifter_2_in := StateOk;
END_TRANSITION
STEP Lifter_2_in:
	Lifter_2_in_action(N);
END_STEP
TRANSITION FROM Lifter_2_in TO Depalletizing_end := StateOk;
END_TRANSITION
STEP Depalletizing_end:
END_STEP
TRANSITION FROM (Palletizing_end, Depalletizing_end) TO SeqEnd := TRUE;
END_TRANSITION
STEP SeqEnd: (* STATE_OK / -> WAIT *)
	SeqEnd_action(N);
END_STEP
TRANSITION FROM SeqEnd TO STATE_WAITForStart := NOT Start;
END_TRANSITION

ACTION Init_action:
Start:=FALSE;
State:=STATE_WAIT;
END_ACTION

ACTION STATE_WAITForStart_action:
IF	Start THEN
	State:=STATE_RUN;
	Result:=RESULT_NON;
	SFCTimeStart:=TIME();
END_IF
END_ACTION

ACTION Belt_down__action:
ST08_404_Y52_0.MoveInit:=TRUE;
END_ACTION

ACTION M_TrayAusheben_unten_entry:
ST08_190_M1.MoveAbs:=TRUE;
ST08_190_M1.Vorgabe_Pos_Abs:=TD.PosTrayAusheben[1].Pos;	(*1=unten, 2=oben, *)
END_ACTION

ACTION Lifter_down__action:
ST08_406_Y52_3.MoveInit:=TRUE;
END_ACTION

ACTION VakuumOff_action:
ST08_403_Y50_6.MoveInit := TRUE;
ST08_403_Y50_7.MoveInit := TRUE;
END_ACTION

ACTION Door2_close_action:
ST08_405_Y51_0.MoveInit:=TRUE;
END_ACTION

ACTION Door3_close_action:
ST08_406_Y51_2.MoveInit:=TRUE;
END_ACTION

ACTION Door4_close_action:
ST08_407_Y51_4.MoveInit:=TRUE;
END_ACTION

ACTION Stopper1_IN_action:
ST08_400_Y50_0.MoveInit:=TRUE; (* Stopper Traystapel Einlaufb. hinten links + rechts AST (Valve) *)
END_ACTION

ACTION Stopper2_IN_action:
ST08_400_Y50_2.MoveInit:=TRUE;
END_ACTION

ACTION Stopper3_IN_action:
ST08_402_Y50_4.MoveInit:=TRUE;
END_ACTION

ACTION schieben1_IN_action:
ST08_401_Y52_4.MoveInit:=TRUE; (*  Traystapel schieben hinten AST (Valve) *)
END_ACTION

ACTION schieben2_IN_action:
ST08_402_Y52_6.MoveInit:=TRUE;
END_ACTION

ACTION schieben3_IN_action:
ST08_402_Y52_7.MoveInit:=TRUE;
END_ACTION

ACTION Stopper_HQE_action:
ST08_404_Y51_6.MoveInit:=TRUE;
END_ACTION

ACTION Check_LifterMotor_entry:
ST08_180_M1.MotorOn:=NOT ST08_180_M1.On;
ST08_185_M1.MotorOn:=NOT ST08_185_M1.On;
END_ACTION

ACTION Aufstapeln_Motor_ein_entry:
ST08_185_M1.Vorgabe_Velo:=1750;
END_ACTION

ACTION Abstapeln_Motor_ein_entry:
ST08_180_M1.Vorgabe_Velo:=1750;
END_ACTION

ACTION FixingOpen_action:
ST08_408_Y54_0.MoveWork:=TRUE;
END_ACTION

ACTION FixingClose_action:
ST08_408_Y54_0.MoveInit:=TRUE;
END_ACTION

ACTION M_Aufstapeln_unten_entry:
ST08_185_M1.MoveAbs:=TRUE;
ST08_185_M1.Vorgabe_Pos_Abs:=TD.PosAufstapeln[1].Pos;	(*1=unten, 2= mitte, 3=oben, 4=frei*)
END_ACTION

ACTION Lifter_1_out_action:
ST08_408_Y54_2.MoveInit:=TRUE;
END_ACTION

ACTION Lifter_2_out_action:
ST08_408_Y54_4.MoveInit:=TRUE;
END_ACTION

ACTION FixingClose__entry:
MP.ST08.NoOfBlisterInStackerOut:=0;
END_ACTION

ACTION FixingClose__action:
ST08_408_Y54_0.MoveInit:=TRUE;
END_ACTION

ACTION Puffer_voll_entry:
MessageHandler.ClearMessageLines(sVisu:=Visu.Message);
END_ACTION

ACTION Puffer_voll_action:
MessageHandler.Msg.ID:='PM201';
MessageHandler.Msg.Name:='St08 Stau im Auslauf';
MessageHandler.Msg.Text:='Auslaufand voll!! Blister entnehmen!!';
MessageHandler.Msg.Color:=Color.blue;
MessageHandler.Msg.Station:=0;


MessageHandler(
	Prio:=2, 							(*1=highest, .. , 4=lowest*)
	Btn1Addr:=ADR(MsgOk),			(*Address of Button1 , if Zero then Button is unvisible*)
	Btn2Addr:=,			(*Address of Button2 , if Zero then Button is unvisible*)
	sVisu:=Visu.Message);
END_ACTION

ACTION Puffer_voll_exit:
MsgOk:=FALSE;
MsgCancel:=FALSE;
END_ACTION

ACTION LifterStopper_Open_action:
ST08_400_Y52_5.MoveWork :=TRUE;
END_ACTION

ACTION LifterStopperDown_action:
ST08_408_Y54_4.MoveInit:=TRUE;
END_ACTION

ACTION BandAusheberWork_action:
ST08_404_Y52_0.MoveWork:=TRUE;
END_ACTION

ACTION Lock4_OPEN_action:
ST08_407_Y51_4.MoveWork:=TRUE;
END_ACTION

ACTION Conveyor_ON_action:
ST08_Palletizing.ConveyorOn:=TRUE;
END_ACTION

ACTION Wait_B55_5_low_entry:
ProcessMessage01:='';
END_ACTION

ACTION Wait_B55_5_low_action:
ProcessMessage01:='1IM12';(*'St. 8 warte Tray ausgelaufen*)
END_ACTION

ACTION Wait_B55_5_low_exit:
ProcessMessage01:='';
END_ACTION

ACTION Wait_B55_5_high_entry:
ProcessMessage01:='';
END_ACTION

ACTION Wait_B55_5_high_action:
ProcessMessage01:='1IM13';(*St. 8 warte Tray auf Rollenbahn*)
END_ACTION

ACTION Lock4_CLOSE_31_action:
ST08_407_Y51_4.MoveInit:=TRUE;
END_ACTION

ACTION Wait_DoorClose_31_entry:
ProcessMessage01:='';
END_ACTION

ACTION Wait_DoorClose_31_action:
ProcessMessage01:='1IM14';(*'St.8 warte Türe 4 auslauf geschlossen*)
END_ACTION

ACTION Wait_DoorClose_31_exit:
ProcessMessage01:='';
END_ACTION

ACTION BandAusheberInit_action:
ST08_404_Y52_0.MoveInit:=TRUE;
END_ACTION

ACTION Conveyor_OFF_action:
ST08_Palletizing.ConveyorOn:=FALSE;
END_ACTION

ACTION LifterStopper_CLOSE_action:
ST08_400_Y52_5.MoveInit:=TRUE;
END_ACTION

ACTION LifterStopperUp__action:
ST08_408_Y54_4.MoveWork:=TRUE;
END_ACTION

ACTION Stopper_in_action:
ST08_400_Y52_5.MoveWork:=TRUE;
END_ACTION

ACTION M_Abstapeln_unten_entry:
ST08_180_M1.MoveAbs:=TRUE;
ST08_180_M1.Vorgabe_Pos_Abs:=TD.PosAbstapeln[1].Pos;	(*1=unten, 2= mitte, 3=oben, 4=frei*)
END_ACTION

ACTION Lifter_1_in_action:
ST08_404_Y53_0.MoveInit:=TRUE;
END_ACTION

ACTION Lifter_2_in_action:
ST08_404_Y53_2.MoveInit:=TRUE;
END_ACTION

ACTION SeqEnd_action:
IF	ST08_406_B54_3.BitInToCheck THEN
	ST08_CallPRGs.PosIdxHelp:=0;
END_IF

IF 	State=STATE_RUN THEN
	SFCTime:=TIME_TO_DINT(TIME()-SFCTimeStart);
	State:=STATE_OK;
END_IF

IF 	NOT Start THEN
	State:=STATE_WAIT;
END_IF
END_ACTION

TRANSITION StateOk:
ST08_404_Y52_0.State=STATE_OK
END_TRANSITION

TRANSITION with_Motor:
MP.ST08.TrayAushebenMotor
END_TRANSITION

TRANSITION busy:
ST08_190_M1.Busy
END_TRANSITION

TRANSITION Done:
ST08_190_M1.Done
END_TRANSITION

TRANSITION StateOk:
ST08_406_Y52_3.State=STATE_OK
END_TRANSITION

TRANSITION VakuumOff:
ST08_403_Y50_6.State=STATE_OK AND
ST08_403_Y50_7.State=STATE_OK
END_TRANSITION

TRANSITION StateOk:
ST08_405_Y51_0.State=STATE_OK
END_TRANSITION

TRANSITION StateOk:
ST08_406_Y51_2.State=STATE_OK
END_TRANSITION

TRANSITION StateOk:
ST08_407_Y51_4.State=STATE_OK
END_TRANSITION

TRANSITION mit Verlaengerung:
MP.ST08.Trayzufuhr_Verlaengerung
END_TRANSITION

TRANSITION #StateOk:
ST08_400_Y50_0.State=STATE_OK
END_TRANSITION

TRANSITION #StateOk:
ST08_400_Y50_2.State=STATE_OK
END_TRANSITION

TRANSITION #StateOk:
ST08_402_Y50_4.State=STATE_OK
END_TRANSITION

TRANSITION mit_schieben:
MP.ST08.Traystapel_schieben
END_TRANSITION

TRANSITION mit Verlaengerung:
MP.ST08.Trayzufuhr_Verlaengerung
END_TRANSITION

TRANSITION #StateOk:
ST08_401_Y52_4.State=STATE_OK
END_TRANSITION

TRANSITION #StateOk:
ST08_402_Y52_6.State=STATE_OK
END_TRANSITION

TRANSITION #StateOk:
ST08_402_Y52_7.State=STATE_OK
END_TRANSITION

TRANSITION StateOk:
ST08_404_Y51_6.State=STATE_OK
END_TRANSITION

TRANSITION with_Motor:
MP.ST08.StapelMotor
END_TRANSITION

TRANSITION Check_LifterMotor:
NOT ST08_180_M1.Error_ AND
ST08_180_M1.On AND
NOT ST08_185_M1.Error_ AND
ST08_185_M1.On
END_TRANSITION

TRANSITION on:
ST08_180_M1.on AND
ST08_185_M1.on
END_TRANSITION

TRANSITION MoveOut:
ST08_Palletizing.MoveOut
END_TRANSITION

TRANSITION StateOk:
ST08_408_Y54_0.State=STATE_OK
END_TRANSITION

TRANSITION StateOk:
ST08_408_Y54_0.State=STATE_OK
END_TRANSITION

TRANSITION with_Motor:
MP.ST08.StapelMotor
END_TRANSITION

TRANSITION MotorOn:
ST08_185_M1.On
END_TRANSITION

TRANSITION busy:
ST08_185_M1.Busy
END_TRANSITION

TRANSITION Done:
ST08_185_M1.Done
END_TRANSITION

TRANSITION StateOk:
ST08_408_Y54_2.State=STATE_OK
END_TRANSITION

TRANSITION StateOk:
ST08_408_Y54_4.State=STATE_OK
END_TRANSITION

TRANSITION NOT_MoveOut:
NOT ST08_Palletizing.MoveOut
END_TRANSITION

TRANSITION NoBlister:
ST08_407_B55_4.BitInToCheck (* Tray in Aufstapelposition eingelaufen STN8 *)
END_TRANSITION

TRANSITION StateOk:
ST08_408_Y54_0.State=STATE_OK
END_TRANSITION

TRANSITION TrayKompletOut:
ST08_409_B55_5.BitInToCheck
END_TRANSITION

